(*!
<summary>Checks percentage dispersion for both signs and bound forwarding.</summary>
<description>
Owns a generator used by one PLC task. Each run checks the same bounds against fresh samples.
The runner binds assertions to the instance address. Keep the instance at that address for its run.
</description>
*)

{attribute 'no_assign'}
{attribute 'no_explicit_call' := 'do not call this function block directly'}
FUNCTION_BLOCK RandomPercentageDispersionTest EXTENDS TOF_Testing.SingleCycleTest
VAR_STAT
	{attribute 'hide'}
	_ClassName : STRING := __POUNAME();
END_VAR
VAR
	_Random : TOF_Core.Random;
END_VAR

(*!
<summary>Samples positive and negative bases and checks exact outcomes for zero and clamped dispersion.</summary>
<description>
The generated ranges have independently calculated endpoints. Enabled bounds cover deterministic cases
outside the generated interval. The test makes no assumptions about sample sequence or distribution.
</description>
*)
METHOD PROTECTED ExecuteTest
VAR
	value : LREAL;
	i : INT;
END_VAR
value := _Random.GetWithDispersionPercent(baseValue := LREAL#-40.0, dispersionPercent := LREAL#0.0);
Assert.ThatLongReal(
	actual := value,
	message := "Zero percent must return the negative base"
).ToBe(expected := LREAL#-40.0);

value := _Random.GetWithDispersionPercent(
	baseValue := LREAL#80.0,
	dispersionPercent := LREAL#25.0,
	minValue := LREAL#110.0
);
Assert.ThatLongReal(
	actual := value,
	message := "Percentage dispersion must forward the lower bound"
).ToBe(expected := LREAL#110.0);

value := _Random.GetWithDispersionPercent(
	baseValue := LREAL#-40.0,
	dispersionPercent := LREAL#25.0,
	maxValue := LREAL#-60.0
);
Assert.ThatLongReal(
	actual := value,
	message := "Percentage dispersion must forward the upper bound"
).ToBe(expected := LREAL#-60.0);

FOR i := 1 TO 21 DO
	value := _Random.GetWithDispersionPercent(baseValue := LREAL#80.0, dispersionPercent := LREAL#25.0);
	Assert.ThatLongReal(
		actual := value,
		message := "Positive base sample below 60"
	).IsGreaterThanOrEquals(expected := LREAL#60.0);
	Assert.ThatLongReal(
		actual := value,
		message := "Positive base sample above 100"
	).IsLessThanOrEquals(expected := LREAL#100.0);

	value := _Random.GetWithDispersionPercent(baseValue := LREAL#-40.0, dispersionPercent := LREAL#25.0);
	Assert.ThatLongReal(
		actual := value,
		message := "Negative base sample below -50"
	).IsGreaterThanOrEquals(expected := LREAL#-50.0);
	Assert.ThatLongReal(
		actual := value,
		message := "Negative base sample above -30"
	).IsLessThanOrEquals(expected := LREAL#-30.0);
END_FOR
END_METHOD

//! <summary>Borrows the concrete class name. Callers must not modify it.</summary>
{attribute 'monitoring' := 'call'}
PROPERTY ClassName : REFERENCE TO STRING
GET
ClassName REF= _ClassName;
END_GET
END_PROPERTY

//! <summary>Borrows the compiler-initialized namespace name. Callers must not modify it.</summary>
{attribute 'monitoring' := 'call'}
PROPERTY NamespaceName : REFERENCE TO STRING
GET
NamespaceName REF= CurrentNamespace.Name;
END_GET
END_PROPERTY

//! <summary>Reports the concrete instance size in bytes.</summary>
{attribute 'monitoring' := 'call'}
PROPERTY SelfSize : ULINT
GET
SelfSize := XSIZEOF(THIS^);
END_GET
END_PROPERTY

END_FUNCTION_BLOCK

// ---- Tests/Core/ExceptionTestGroup.TcPOU
(*
SPDX-FileCopyrightText: c 2026 Oleksandr Tiutyk <trofimich@gmail.com>
SPDX-License-Identifier: MIT
License: https://opensource.org/license/mit
*)

(*!
<summary>Groups exception transport, diagnostics, cloning and graph contract tests.</summary>
<description>
Owns the independent child instances and their fixed registration array. Use from one PLC task at a stable address.
</description>
*)

{attribute 'no_assign'}
{attribute 'no_explicit_call' := 'do not call this function block directly'}
FUNCTION_BLOCK ExceptionTestGroup EXTENDS TOF_Testing.TestGroup<12>
VAR_STAT
	{attribute 'hide'}
	_ClassName : STRING := __POUNAME();
END_VAR
VAR
	_NotImplemented : NotImplementedExceptionTest(name := "SimpleException", parent := THIS^);
	_StandardChain : StandardExceptionChainTest(name := "StandardExceptions", parent := THIS^);
	_Aggregate : AggregateExceptionPropagationTest(name := "AggregateException", parent := THIS^);
	_SavedFramework : SavedFrameworkExceptionRethrowTest(name := "RethrowSavedFrameworkException", parent := THIS^);
	_NativeRethrow : SystemExceptionRethrowTest(name := "RethrowSystemExceptionAfterFramework", parent := THIS^);
	_TimestampFormatting : ExceptionTimestampFormattingTest(name := "TimestampFormatting", parent := THIS^);
	_SystemTimestamp : SystemExceptionTimestampFormattingTest(
		name := "SystemExceptionTimestampFormatting",
		parent := THIS^
	);
	_SystemClone : SystemExceptionCloneTest(name := "SystemExceptionClone", parent := THIS^);
	_AggregateClone : AggregateExceptionCloneTest(name := "AggregateCloneLifetime", parent := THIS^);
	_ArgumentTypeClone : ArgumentTypeExceptionCloneTest(name := "ArgumentTypeCloneIdentity", parent := THIS^);
	_GraphRejection : ExceptionGraphRejectionTest(name := "GraphRejection", parent := THIS^);
	_BoundedMessage : AggregateExceptionBoundedMessageTest(name := "BoundedMessage", parent := THIS^);

	_Children : ARRAY [0.._ChildCount - 1] OF TOF_Testing.ITestElement :=
	[
		_NotImplemented,
		_StandardChain,
		_Aggregate,
		_SavedFramework,
		_NativeRethrow,
		_TimestampFormatting,
		_SystemTimestamp,
		_SystemClone,
		_AggregateClone,
		_ArgumentTypeClone,
		_GraphRejection,
		_BoundedMessage
	];
END_VAR

//! <summary>Borrows the fixed child array. Callers must not modify it.</summary>
{attribute 'monitoring' := 'call'}
PROPERTY Children : REFERENCE TO ARRAY [0.._ChildCount - 1] OF TOF_Testing.ITestElement
GET
Children REF= _Children;
END_GET
END_PROPERTY

//! <summary>Borrows the concrete class name. Callers must not modify it.</summary>
{attribute 'monitoring' := 'call'}
PROPERTY ClassName : REFERENCE TO STRING
GET
ClassName REF= _ClassName;
END_GET
END_PROPERTY

//! <summary>Borrows the compiler-initialized namespace name. Callers must not modify it.</summary>
{attribute 'monitoring' := 'call'}
PROPERTY NamespaceName : REFERENCE TO STRING
GET
NamespaceName REF= CurrentNamespace.Name;
END_GET
END_PROPERTY

//! <summary>Reports the concrete instance size in bytes.</summary>
{attribute 'monitoring' := 'call'}
PROPERTY SelfSize : ULINT
GET
SelfSize := XSIZEOF(THIS^);
END_GET
END_PROPERTY

END_FUNCTION_BLOCK

// ---- Tests/Core/NotImplementedExceptionTest.TcPOU
(*
SPDX-FileCopyrightText: c 2026 Oleksandr Tiutyk <trofimich@gmail.com>
SPDX-License-Identifier: MIT
License: https://opensource.org/license/mit
*)

(*!
<summary>Checks concrete exception transport and diagnostics for an unimplemented POU.</summary>
<description>
Uses one task and stays at a stable address while assertions are bound to this instance.
</description>
*)

{attribute 'no_assign'}
{attribute 'no_explicit_call' := 'do not call this function block directly'}
FUNCTION_BLOCK NotImplementedExceptionTest EXTENDS TOF_Testing.SingleCycleTest
VAR_STAT
	{attribute 'hide'}
	_ClassName : STRING := __POUNAME();
END_VAR

(*!
<summary>Checks concrete exception transport and diagnostics for an unimplemented POU.</summary>
<description>
Injects a fixed source location so the expected text and metadata are independent of this test's name.
</description>
*)
METHOD PROTECTED ExecuteTest
VAR
	exceptionCode : __SYSTEM.ExceptionCode;
	caught : TOF_Core.IException;
	typed : TOF_Core.INotImplementedException;
	message : TOF_Core.ERROR_MESSAGE;
END_VAR
// Raise one exception to exercise the transport from the facade to the catch.
__TRY
	TOF_Core.Exceptions.ThrowNotImplemented(
		sourceNamespaceName := 'Tests',
		sourceClassName := 'ExceptionFixture',
		sourcePOUName := 'UnimplementedOperation',
		sourcePosition := 'P1'
	);
__CATCH(exceptionCode)
	caught := TOF_Core.ExceptionManager.GetLastException(
		exceptionCode := exceptionCode,
		catchPointNamespaceName := NamespaceName,
		catchPointPOUName := __POUNAME(),
		catchPointPosition := __POSITION()
	);
__ENDTRY

IF NOT __QUERYINTERFACE(caught, typed) THEN
	RecordFailure(message := "ThrowNotImplemented must propagate NotImplementedException");
	RETURN;
END_IF

message := typed.GetMessage();
Assert.ThatBool(
	actual := message = "Program organization unit 'Tests.ExceptionFixture.UnimplementedOperation()' is not implemented",
	message := "NotImplementedException must name the supplied POU"
).IsTrue();
Assert.ThatBool(
	actual := typed.SourcePosition = 'P1',
	message := "NotImplementedException must preserve the throw position"
).IsTrue();
Assert.ThatBool(
	actual := typed.IsDynamicInstance,
	message := "Facade transport must yield a task-managed exception"
).IsTrue();
END_METHOD

//! <summary>Borrows the concrete class name. Callers must not modify it.</summary>
{attribute 'monitoring' := 'call'}
PROPERTY ClassName : REFERENCE TO STRING
GET
ClassName REF= _ClassName;
END_GET
END_PROPERTY

//! <summary>Borrows the compiler-initialized namespace name. Callers must not modify it.</summary>
{attribute 'monitoring' := 'call'}
PROPERTY NamespaceName : REFERENCE TO STRING
GET
NamespaceName REF= CurrentNamespace.Name;
END_GET
END_PROPERTY

//! <summary>Reports the concrete instance size in bytes.</summary>
{attribute 'monitoring' := 'call'}
PROPERTY SelfSize : ULINT
GET
SelfSize := XSIZEOF(THIS^);
END_GET
END_PROPERTY

END_FUNCTION_BLOCK

// ---- Tests/Core/StandardExceptionChainTest.TcPOU
(*
SPDX-FileCopyrightText: c 2026 Oleksandr Tiutyk <trofimich@gmail.com>
SPDX-License-Identifier: MIT
License: https://opensource.org/license/mit
*)

(*!
<summary>Checks the text, inner identity and root of a three-level standard exception chain.</summary>
<description>
Uses one task and stays at a stable address while assertions are bound to this instance.
</description>
*)

{attribute 'no_assign'}
{attribute 'no_explicit_call' := 'do not call this function block directly'}
FUNCTION_BLOCK StandardExceptionChainTest EXTENDS TOF_Testing.SingleCycleTest
VAR_STAT
	{attribute 'hide'}
	_ClassName : STRING := __POUNAME();
END_VAR

(*!
<summary>Checks the text, inner identity and root of a three-level standard exception chain.</summary>
<description>
Keeps only cycle-local references. Compares the root with the first caught cause through read-only views.
ToError copies the outer diagnostic and the deepest cause.
</description>
*)
METHOD PROTECTED ExecuteTest
VAR
	exceptionCode : __SYSTEM.ExceptionCode;
	caught : TOF_Core.IException;
	previous : TOF_Core.IException;
	previousView : TOF_Core.IReadOnlyException;
	first : TOF_Core.IReadOnlyException;
	root : TOF_Core.IReadOnlyException;
	typed : TOF_Core.IStandardException;

	inputs : ARRAY [0..2] OF WSTRING := ["First cause", "Second cause", "Outer failure"];
	expected : ARRAY [0..2] OF WSTRING := [
		"First cause",
		"Second cause -> First cause",
		"Outer failure -> Second cause -> First cause"
	];
	message : TOF_Core.ERROR_MESSAGE;
	actual : TOF_Core.ERROR_MESSAGE;
	snapshot : TOF_Core.ERROR;
	i : DINT;
END_VAR
FOR i := 0 TO UPPER_BOUND(inputs, 1) DO
	message := inputs[i];
	caught := 0;

	// Each deliberate throw adds one outer cause and is captured before asserting its payload.
	__TRY
		TOF_Core.Exceptions.ThrowStandard(
			sourceNamespaceName := NamespaceName,
			sourceClassName := ClassName,
			sourcePOUName := __POUNAME(),
			sourcePosition := __POSITION(),
			message := message,
			innerException := previous
		);
	__CATCH(exceptionCode)
		caught := TOF_Core.ExceptionManager.GetLastException(
			exceptionCode := exceptionCode,
			catchPointNamespaceName := NamespaceName,
			catchPointPOUName := __POUNAME(),
			catchPointPosition := __POSITION()
		);
	__ENDTRY

	IF NOT __QUERYINTERFACE(caught, typed) THEN
		Assert.ThatBool(
			actual := FALSE,
			message := Tc2_Utilities.WCONCAT(STR1 := "StandardException missing for ", STR2 := inputs[i])
		).IsTrue();
		RETURN;
	END_IF

	actual := typed.GetMessage();
	Assert.ThatBool(
		actual := actual = expected[i],
		message := Tc2_Utilities.WCONCAT(STR1 := "Incorrect chain text for ", STR2 := inputs[i])
	).IsTrue();
	Assert.ThatBool(
		actual := typed.InnerException = previousView,
		message := Tc2_Utilities.WCONCAT(STR1 := "Incorrect immediate cause for ", STR2 := inputs[i])
	).IsTrue();

	IF i = 0 THEN
		first := typed;
	END_IF

	previous := caught;
	previousView := typed;
END_FOR

root := typed.GetRootException();
Assert.ThatBool(
	actual := root = first,
	message := "The outer standard exception must reach the first cause"
).IsTrue();
typed.ToError(targetError := snapshot, severity := TOF_Core.ERROR_SEVERITY.CRITICAL);
Assert.ThatBool(
	actual := snapshot.TopMessage = expected[2] AND_THEN snapshot.RootMessage = "First cause",
	message := "The ERROR snapshot must keep the outer diagnostics and the deepest cause"
).IsTrue();
Assert.ThatBool(
	actual := snapshot.Severity = TOF_Core.ERROR_SEVERITY.CRITICAL,
	message := "ToError must copy the supplied severity"
).IsTrue();
END_METHOD

//! <summary>Borrows the concrete class name. Callers must not modify it.</summary>
{attribute 'monitoring' := 'call'}
PROPERTY ClassName : REFERENCE TO STRING
GET
ClassName REF= _ClassName;
END_GET
END_PROPERTY

//! <summary>Borrows the compiler-initialized namespace name. Callers must not modify it.</summary>
{attribute 'monitoring' := 'call'}
PROPERTY NamespaceName : REFERENCE TO STRING
GET
NamespaceName REF= CurrentNamespace.Name;
END_GET
END_PROPERTY

//! <summary>Reports the concrete instance size in bytes.</summary>
{attribute 'monitoring' := 'call'}
PROPERTY SelfSize : ULINT
GET
SelfSize := XSIZEOF(THIS^);
END_GET
END_PROPERTY

END_FUNCTION_BLOCK

// ---- Tests/Core/AggregateExceptionPropagationTest.TcPOU
(*
SPDX-FileCopyrightText: c 2026 Oleksandr Tiutyk <trofimich@gmail.com>
SPDX-License-Identifier: MIT
License: https://opensource.org/license/mit
*)

(*!
<summary>Checks aggregate flattening, transport, ordering and diagnostic snapshots.</summary>
<description>
Uses one task and stays at a stable address while assertions are bound to this instance.
</description>
*)

{attribute 'no_assign'}
{attribute 'no_explicit_call' := 'do not call this function block directly'}
FUNCTION_BLOCK AggregateExceptionPropagationTest EXTENDS TOF_Testing.SingleCycleTest
VAR_STAT
	{attribute 'hide'}
	_ClassName : STRING := __POUNAME();
END_VAR
VAR
	_Aggregate : TOF_Core.AggregateException;
	_AdditionalCauses : TOF_Core.AggregateException;
END_VAR

(*!
<summary>Checks aggregate flattening, transport, ordering and diagnostic snapshots.</summary>
<description>
The persistent arrays belong to this test. Within the current PLC cycle, compares borrowed causes by
read-only interface identity and checks null results on both sides of the valid index range.
Compares the full default message and reports the expected and actual text if they differ.
</description>
*)
METHOD PROTECTED ExecuteTest
VAR
	exceptionCode : __SYSTEM.ExceptionCode;
	caught : TOF_Core.IException;
	cause : TOF_Core.IStandardException;
	aggregate : TOF_Core.IAggregateException;
	causes : ARRAY [0..2] OF TOF_Core.IReadOnlyException;
	observedCause : TOF_Core.IReadOnlyException;

	causeMessages : ARRAY [0..2] OF WSTRING := ["First cause", "Second cause", "Third cause"];
	causeMessage : TOF_Core.ERROR_MESSAGE;
	message : TOF_Core.ERROR_MESSAGE;
	expectedMessage : TOF_Core.ERROR_MESSAGE;
	snapshot : TOF_Core.ERROR;
	i : DINT;
END_VAR
FOR i := 0 TO UPPER_BOUND(causes, 1) DO
	causeMessage := causeMessages[i];
	caught := 0;

	// Capture each deliberate throw before adding its task-owned payload to the fixture.
	__TRY
		TOF_Core.Exceptions.ThrowStandard(
			sourceNamespaceName := NamespaceName,
			sourceClassName := ClassName,
			sourcePOUName := 'RaiseCause',
			sourcePosition := __POSITION(),
			message := causeMessage
		);
	__CATCH(exceptionCode)
		caught := TOF_Core.ExceptionManager.GetLastException(
			exceptionCode := exceptionCode,
			catchPointNamespaceName := NamespaceName,
			catchPointPOUName := __POUNAME(),
			catchPointPosition := __POSITION()
		);
	__ENDTRY

	IF NOT __QUERYINTERFACE(caught, cause) THEN
		Assert.ThatBool(
			actual := FALSE,
			message := Tc2_Utilities.WCONCAT(STR1 := "Aggregate setup did not catch ", STR2 := causeMessages[i])
		).IsTrue();
		RETURN;
	END_IF

	causes[i] := cause;

	IF i = 0 THEN
		_Aggregate.AddInnerException(innerException := cause);
	ELSE
		_AdditionalCauses.AddInnerException(innerException := cause);
	END_IF
END_FOR

_Aggregate.AddInnerException(innerException := _AdditionalCauses);
_AdditionalCauses.Clear();

// Catch the aggregate snapshot before clearing its caller-owned source.
caught := 0;

__TRY
	_Aggregate.Throw(
		sourceNamespaceName := NamespaceName,
		sourceClassName := ClassName,
		sourcePOUName := __POUNAME(),
		sourcePosition := __POSITION()
	);
__CATCH(exceptionCode)
	caught := TOF_Core.ExceptionManager.GetLastException(
		exceptionCode := exceptionCode,
		catchPointNamespaceName := NamespaceName,
		catchPointPOUName := __POUNAME(),
		catchPointPosition := __POSITION()
	);
__ENDTRY

_Aggregate.Clear();

IF NOT __QUERYINTERFACE(caught, aggregate) THEN
	RecordFailure(message := "Aggregate Throw must propagate a concrete aggregate snapshot");
	RETURN;
END_IF

Assert.ThatUInt(
	actual := aggregate.InnerExceptionCount,
	message := "The propagated aggregate must contain all three flattened causes"
).ToBe(expected := UINT#3);

FOR i := 0 TO UPPER_BOUND(causes, 1) DO
	observedCause := aggregate.GetInnerException(index := i);
	Assert.ThatBool(
		actual := observedCause = causes[i],
		message := Tc2_Utilities.WCONCAT(STR1 := "Wrong aggregate position for ", STR2 := causeMessages[i])
	).IsTrue();
END_FOR

observedCause := aggregate.GetInnerException(index := -1);
Assert.ThatBool(
	actual := observedCause = 0,
	message := "Aggregate indexing before the first entry must return null"
).IsTrue();

observedCause := aggregate.GetInnerException(index := 3);
Assert.ThatBool(
	actual := observedCause = 0,
	message := "Aggregate indexing after the last entry must return null"
).IsTrue();

observedCause := aggregate.GetRootException();
Assert.ThatBool(
	actual := observedCause = causes[0],
	message := "Aggregate root must come from the first cause"
).IsTrue();

// The index suffix includes a space and the formatter appends one more before each cause.
expectedMessage := "3 aggregated exceptions$R0:  First cause$R1:  Second cause$R2:  Third cause";
message := aggregate.GetMessage();
Assert.That(
	actual := message,
	message := "The aggregate must describe all three causes in index order"
).ToBe(expected := expectedMessage);

aggregate.ToError(targetError := snapshot, severity := TOF_Core.ERROR_SEVERITY.CRITICAL);
Assert.ThatBool(
	actual := snapshot.TopMessage = message AND_THEN snapshot.RootMessage = "First cause",
	message := "The aggregate ERROR must copy the complete message and the first root diagnostic"
).IsTrue();
Assert.ThatBool(
	actual := snapshot.Severity = TOF_Core.ERROR_SEVERITY.CRITICAL,
	message := "Aggregate ToError must copy the supplied severity"
).IsTrue();
END_METHOD

(*!
<summary>Clears the caller-owned aggregate storage before the result is reported.</summary>
<description>
Safe after partial setup or repeated Clear. The task memory manager retains ownership of dynamic causes.
</description>
*)
METHOD PROTECTED AfterTest
_AdditionalCauses.Clear();
_Aggregate.Clear();
END_METHOD

//! <summary>Borrows the concrete class name. Callers must not modify it.</summary>
{attribute 'monitoring' := 'call'}
PROPERTY ClassName : REFERENCE TO STRING
GET
ClassName REF= _ClassName;
END_GET
END_PROPERTY

//! <summary>Borrows the compiler-initialized namespace name. Callers must not modify it.</summary>
{attribute 'monitoring' := 'call'}
PROPERTY NamespaceName : REFERENCE TO STRING
GET
NamespaceName REF= CurrentNamespace.Name;
END_GET
END_PROPERTY

//! <summary>Reports the concrete instance size in bytes.</summary>
{attribute 'monitoring' := 'call'}
PROPERTY SelfSize : ULINT
GET
SelfSize := XSIZEOF(THIS^);
END_GET
END_PROPERTY

END_FUNCTION_BLOCK

// ---- Tests/Core/SavedFrameworkExceptionRethrowTest.TcPOU
(*
SPDX-FileCopyrightText: c 2026 Oleksandr Tiutyk <trofimich@gmail.com>
SPDX-License-Identifier: MIT
License: https://opensource.org/license/mit
*)

(*!
<summary>Checks rethrow of a saved framework payload after a different nested exception.</summary>
<description>
Uses one task and stays at a stable address while assertions are bound to this instance.
</description>
*)

{attribute 'no_assign'}
{attribute 'no_explicit_call' := 'do not call this function block directly'}
FUNCTION_BLOCK SavedFrameworkExceptionRethrowTest EXTENDS TOF_Testing.SingleCycleTest
VAR_STAT
	{attribute 'hide'}
	_ClassName : STRING := __POUNAME();
END_VAR

(*!
<summary>Checks rethrow of a saved framework payload after a different nested exception.</summary>
<description>
The nested handler must capture its own payload. All caught references are used only in the current task cycle.
</description>
*)
METHOD PROTECTED ExecuteTest
VAR
	exceptionCode : __SYSTEM.ExceptionCode;
	saved : TOF_Core.IException;
	outerCode : __SYSTEM.ExceptionCode;
	nestedCode : __SYSTEM.ExceptionCode;
	nested : TOF_Core.IException;
	received : TOF_Core.IException;
	nestedMessage : TOF_Core.ERROR_MESSAGE;
	receivedMessage : TOF_Core.ERROR_MESSAGE;
END_VAR
// Catch the original, let a nested handler replace the active payload, then rethrow the saved object.
__TRY
	__TRY
		TOF_Core.Exceptions.ThrowStandard(
			sourceNamespaceName := NamespaceName,
			sourceClassName := ClassName,
			sourcePOUName := __POUNAME(),
			sourcePosition := __POSITION(),
			message := "Original"
		);
	__CATCH(exceptionCode)
		saved := TOF_Core.ExceptionManager.GetLastException(
			exceptionCode := exceptionCode,
			catchPointNamespaceName := NamespaceName,
			catchPointPOUName := __POUNAME(),
			catchPointPosition := __POSITION()
		);

		__TRY
			TOF_Core.Exceptions.ThrowStandard(
				sourceNamespaceName := NamespaceName,
				sourceClassName := ClassName,
				sourcePOUName := __POUNAME(),
				sourcePosition := __POSITION(),
				message := "Nested"
			);
		__CATCH(nestedCode)
			nested := TOF_Core.ExceptionManager.GetLastException(
				exceptionCode := nestedCode,
				catchPointNamespaceName := NamespaceName,
				catchPointPOUName := __POUNAME(),
				catchPointPosition := __POSITION()
			);
		__ENDTRY

		IF saved <> 0 THEN
			TOF_Core.ExceptionManager.Throw(exception := saved);
		END_IF
	__ENDTRY
__CATCH(outerCode)
	received := TOF_Core.ExceptionManager.GetLastException(
		exceptionCode := outerCode,
		catchPointNamespaceName := NamespaceName,
		catchPointPOUName := __POUNAME(),
		catchPointPosition := __POSITION()
	);
__ENDTRY

IF nested = 0 OR_ELSE received = 0 THEN
	RecordFailure(message := "The nested throw and the saved rethrow must both reach their handlers");
	RETURN;
END_IF

nestedMessage := nested.GetMessage();
receivedMessage := received.GetMessage();
Assert.ThatBool(
	actual := nested <> saved AND_THEN nestedMessage = "Nested",
	message := "The nested catch must observe a distinct payload"
).IsTrue();
Assert.ThatBool(
	actual := received = saved AND_THEN receivedMessage = "Original",
	message := "Rethrow must preserve the saved payload and text"
).IsTrue();
END_METHOD

//! <summary>Borrows the concrete class name. Callers must not modify it.</summary>
{attribute 'monitoring' := 'call'}
PROPERTY ClassName : REFERENCE TO STRING
GET
ClassName REF= _ClassName;
END_GET
END_PROPERTY

//! <summary>Borrows the compiler-initialized namespace name. Callers must not modify it.</summary>
{attribute 'monitoring' := 'call'}
PROPERTY NamespaceName : REFERENCE TO STRING
GET
NamespaceName REF= CurrentNamespace.Name;
END_GET
END_PROPERTY

//! <summary>Reports the concrete instance size in bytes.</summary>
{attribute 'monitoring' := 'call'}
PROPERTY SelfSize : ULINT
GET
SelfSize := XSIZEOF(THIS^);
END_GET
END_PROPERTY

END_FUNCTION_BLOCK

// ---- Tests/Core/SystemExceptionRethrowTest.TcPOU
(*
SPDX-FileCopyrightText: c 2026 Oleksandr Tiutyk <trofimich@gmail.com>
SPDX-License-Identifier: MIT
License: https://opensource.org/license/mit
*)

(*!
<summary>Checks native wrapper propagation through both framework rethrow APIs.</summary>
<description>
Uses one task and stays at a stable address while assertions are bound to this instance.
</description>
*)

{attribute 'no_assign'}
{attribute 'no_explicit_call' := 'do not call this function block directly'}
FUNCTION_BLOCK SystemExceptionRethrowTest EXTENDS TOF_Testing.SingleCycleTest
VAR_STAT
	{attribute 'hide'}
	_ClassName : STRING := __POUNAME();
END_VAR

(*!
<summary>Checks native wrapper propagation through both framework rethrow APIs.</summary>
<description>
Models captured native codes. A second native catch overwrites the shared wrapper while the propagated
snapshot retains its identity and payload until task cleanup.
</description>
*)
METHOD PROTECTED ExecuteTest
VAR
	exceptionCode : __SYSTEM.ExceptionCode;
	frameworkException : TOF_Core.IException;
	original : TOF_Core.IException;
	received : TOF_Core.IException;
	repeated : TOF_Core.IException;
	other : TOF_Core.IException;
	otherWrapper : TOF_Core.ISystemException;
	firstWrapper : TOF_Core.ISystemException;
	codeOnlyWrapper : TOF_Core.ISystemException;
	originalMessage : TOF_Core.ERROR_MESSAGE;
	message : TOF_Core.ERROR_MESSAGE;
	localTimestamp : LDATE_AND_TIME;
	utcTimestamp : LDATE_AND_TIME;
END_VAR
// Establish a framework payload before supplying an already received native code.
__TRY
	TOF_Core.Exceptions.ThrowStandard(
		sourceNamespaceName := NamespaceName,
		sourceClassName := ClassName,
		sourcePOUName := __POUNAME(),
		sourcePosition := __POSITION(),
		message := "Earlier framework payload"
	);
__CATCH(exceptionCode)
	frameworkException := TOF_Core.ExceptionManager.GetLastException(
		exceptionCode := exceptionCode,
		catchPointNamespaceName := NamespaceName,
		catchPointPOUName := __POUNAME(),
		catchPointPosition := __POSITION()
	);
__ENDTRY

IF frameworkException = 0 THEN
	RecordFailure(message := "The earlier framework throw must reach its handler");
	RETURN;
END_IF

original := TOF_Core.ExceptionManager.GetLastException(
	exceptionCode := __SYSTEM.ExceptionCode.RTSEXCPT_ARRAYBOUNDS,
	catchPointNamespaceName := 'Tests',
	catchPointPOUName := 'OriginalCatch',
	catchPointPosition := 'P1'
);

IF original = 0 THEN
	RecordFailure(message := "The captured native code must provide a wrapper");
	RETURN;
END_IF

originalMessage := original.GetMessage();
localTimestamp := original.LocalTimestamp;
utcTimestamp := original.UtcTimestamp;

// Transport the static native wrapper as a task-managed framework payload.
__TRY
	TOF_Core.ExceptionManager.Throw(exception := original);
__CATCH(exceptionCode)
	received := TOF_Core.ExceptionManager.GetLastException(
		exceptionCode := exceptionCode,
		catchPointNamespaceName := NamespaceName,
		catchPointPOUName := __POUNAME(),
		catchPointPosition := __POSITION()
	);
__ENDTRY

IF NOT __QUERYINTERFACE(received, firstWrapper) THEN
	RecordFailure(message := "Throw must preserve ISystemException after an earlier framework exception");
	RETURN;
END_IF

Assert.ThatBool(
	actual := firstWrapper.IsDynamicInstance AND_THEN received <> original,
	message := "Native propagation must clone the shared static wrapper"
).IsTrue();
Assert.ThatBool(
	actual := firstWrapper.ExceptionCode = __SYSTEM.ExceptionCode.RTSEXCPT_ARRAYBOUNDS,
	message := "The propagated wrapper must retain its captured native code"
).IsTrue();
Assert.ThatBool(
	actual := firstWrapper.LocalTimestamp = localTimestamp AND_THEN firstWrapper.UtcTimestamp = utcTimestamp,
	message := "Propagation must preserve both original timestamps"
).IsTrue();

other := TOF_Core.ExceptionManager.GetLastException(
	exceptionCode := __SYSTEM.ExceptionCode.RTSEXCPT_ACCESS_VIOLATION,
	catchPointNamespaceName := 'Tests',
	catchPointPOUName := 'OtherCatch',
	catchPointPosition := 'P2'
);
Assert.ThatBool(
	actual := other = original,
	message := "Another native catch must reuse the task wrapper"
).IsTrue();
Assert.ThatBool(
	actual := __QUERYINTERFACE(other, otherWrapper)
		AND_THEN otherWrapper.ExceptionCode = __SYSTEM.ExceptionCode.RTSEXCPT_ACCESS_VIOLATION,
	message := "The shared wrapper must actually observe the later native code"
).IsTrue();

message := firstWrapper.GetMessage();
Assert.ThatBool(
	actual := message = originalMessage
		AND_THEN Tc2_Standard.WFIND(STR1 := message, STR2 := "Tests.OriginalCatch at P1") > 0,
	message := "The propagated wrapper must keep its original diagnostic after the shared wrapper is overwritten"
).IsTrue();

// Replace the manager payload before rethrowing the saved dynamic wrapper.
frameworkException := 0;

__TRY
	TOF_Core.Exceptions.ThrowStandard(
		sourceNamespaceName := NamespaceName,
		sourceClassName := ClassName,
		sourcePOUName := __POUNAME(),
		sourcePosition := __POSITION(),
		message := "Intervening framework payload"
	);
__CATCH(exceptionCode)
	frameworkException := TOF_Core.ExceptionManager.GetLastException(
		exceptionCode := exceptionCode,
		catchPointNamespaceName := NamespaceName,
		catchPointPOUName := __POUNAME(),
		catchPointPosition := __POSITION()
	);
__ENDTRY

Assert.ThatBool(
	actual := frameworkException <> 0 AND_THEN frameworkException <> received,
	message := "An intervening framework throw must install a different payload"
).IsTrue();

__TRY
	TOF_Core.ExceptionManager.Throw(exception := received);
__CATCH(exceptionCode)
	repeated := TOF_Core.ExceptionManager.GetLastException(
		exceptionCode := exceptionCode,
		catchPointNamespaceName := NamespaceName,
		catchPointPOUName := __POUNAME(),
		catchPointPosition := __POSITION()
	);
__ENDTRY

Assert.ThatBool(
	actual := repeated = received,
	message := "Rethrowing the dynamic wrapper must preserve its identity"
).IsTrue();

// Exercise callers that pass a native code and catch point instead of keeping a payload.
repeated := 0;

__TRY
	TOF_Core.ExceptionManager.ReThrowLastException(
		exceptionCode := __SYSTEM.ExceptionCode.RTSEXCPT_ARRAYBOUNDS,
		catchPointNamespaceName := 'Tests',
		catchPointPOUName := 'OriginalCatch',
		catchPointPosition := 'P1'
	);
__CATCH(exceptionCode)
	repeated := TOF_Core.ExceptionManager.GetLastException(
		exceptionCode := exceptionCode,
		catchPointNamespaceName := NamespaceName,
		catchPointPOUName := __POUNAME(),
		catchPointPosition := __POSITION()
	);
__ENDTRY

IF NOT __QUERYINTERFACE(repeated, codeOnlyWrapper) THEN
	RecordFailure(message := "Code-only rethrow must provide an ISystemException payload");
	RETURN;
END_IF

message := codeOnlyWrapper.GetMessage();
Assert.ThatBool(
	actual := message = originalMessage,
	message := "Code-only rethrow must retain the supplied native diagnostic and location"
).IsTrue();
Assert.ThatBool(
	actual := codeOnlyWrapper.ExceptionCode = __SYSTEM.ExceptionCode.RTSEXCPT_ARRAYBOUNDS,
	message := "Code-only rethrow must preserve the native code"
).IsTrue();
END_METHOD

//! <summary>Borrows the concrete class name. Callers must not modify it.</summary>
{attribute 'monitoring' := 'call'}
PROPERTY ClassName : REFERENCE TO STRING
GET
ClassName REF= _ClassName;
END_GET
END_PROPERTY

//! <summary>Borrows the compiler-initialized namespace name. Callers must not modify it.</summary>
{attribute 'monitoring' := 'call'}
PROPERTY NamespaceName : REFERENCE TO STRING
GET
NamespaceName REF= CurrentNamespace.Name;
END_GET
END_PROPERTY

//! <summary>Reports the concrete instance size in bytes.</summary>
{attribute 'monitoring' := 'call'}
PROPERTY SelfSize : ULINT
GET
SelfSize := XSIZEOF(THIS^);
END_GET
END_PROPERTY

END_FUNCTION_BLOCK

// ---- Tests/Core/ExceptionTimestampFormattingTest.TcPOU
(*
SPDX-FileCopyrightText: c 2026 Oleksandr Tiutyk <trofimich@gmail.com>
SPDX-License-Identifier: MIT
License: https://opensource.org/license/mit
*)

(*!
<summary>Checks the shared exception timestamp formatter with fixed local and UTC inputs.</summary>
<description>
Uses one task and stays at a stable address while assertions are bound to this instance.
</description>
*)

{attribute 'no_assign'}
{attribute 'no_explicit_call' := 'do not call this function block directly'}
FUNCTION_BLOCK ExceptionTimestampFormattingTest EXTENDS TOF_Testing.SingleCycleTest
VAR_STAT
	{attribute 'hide'}
	_ClassName : STRING := __POUNAME();
END_VAR
VAR
	_Probe : ExceptionTimestampProbe;
END_VAR

(*!
<summary>Checks the shared exception timestamp formatter with fixed local and UTC inputs.</summary>
<description>
Calls the existing adapter with deterministic timestamps. The result uses the exception diagnostic capacity.
</description>
*)
METHOD PROTECTED ExecuteTest
VAR
	message : TOF_Core.ERROR_MESSAGE;
END_VAR
VAR CONSTANT
	LOCAL_TIMESTAMP : LDATE_AND_TIME := LDT#2026-10-06-15:04:05;
	UTC_TIMESTAMP : LDATE_AND_TIME := LDT#2026-10-06-12:04:05;
END_VAR
message := _Probe.FormatTimestamp(
	mode := TOF_Core.TIMESTAMP_DISPLAY_MODE.HIDDEN,
	localTime := LOCAL_TIMESTAMP,
	utcTime := UTC_TIMESTAMP
);
Assert.ThatBool(
	actual := message = "",
	message := "Hidden timestamp must leave an empty target unchanged"
).IsTrue();

message := _Probe.FormatTimestamp(
	mode := TOF_Core.TIMESTAMP_DISPLAY_MODE.LOCAL,
	localTime := LOCAL_TIMESTAMP,
	utcTime := UTC_TIMESTAMP
);
Assert.ThatBool(
	actual := Tc2_Standard.WFIND(STR1 := message, STR2 := "15:04:05") > 0,
	message := "LOCAL formatting must use local time"
).IsTrue();
Assert.ThatBool(
	actual := Tc2_Standard.WFIND(STR1 := message, STR2 := "UTC") = 0,
	message := "LOCAL formatting must omit the UTC suffix"
).IsTrue();

message := _Probe.FormatTimestamp(
	mode := TOF_Core.TIMESTAMP_DISPLAY_MODE.UTC,
	localTime := LOCAL_TIMESTAMP,
	utcTime := UTC_TIMESTAMP
);
Assert.ThatBool(
	actual := Tc2_Standard.WFIND(STR1 := message, STR2 := "12:04:05") > 0,
	message := "UTC formatting must use UTC time"
).IsTrue();
Assert.ThatBool(
	actual := Tc2_Standard.WRIGHT(STR := message, SIZE := 3) = "UTC",
	message := "UTC formatting must retain the UTC suffix"
).IsTrue();
END_METHOD

//! <summary>Borrows the concrete class name. Callers must not modify it.</summary>
{attribute 'monitoring' := 'call'}
PROPERTY ClassName : REFERENCE TO STRING
GET
ClassName REF= _ClassName;
END_GET
END_PROPERTY

//! <summary>Borrows the compiler-initialized namespace name. Callers must not modify it.</summary>
{attribute 'monitoring' := 'call'}
PROPERTY NamespaceName : REFERENCE TO STRING
GET
NamespaceName REF= CurrentNamespace.Name;
END_GET
END_PROPERTY

//! <summary>Reports the concrete instance size in bytes.</summary>
{attribute 'monitoring' := 'call'}
PROPERTY SelfSize : ULINT
GET
SelfSize := XSIZEOF(THIS^);
END_GET
END_PROPERTY

END_FUNCTION_BLOCK

// ---- Tests/Core/ExceptionTimestampProbe.TcPOU
(*
SPDX-FileCopyrightText: © 2026 Oleksandr Tiutyk <trofimich@gmail.com>
SPDX-License-Identifier: MIT
License: https://opensource.org/license/mit
*)

(*!
<summary>Static test adapter exposing the inherited formatter with deterministic inputs.</summary>
*)

FUNCTION_BLOCK ExceptionTimestampProbe EXTENDS TOF_Core.StandardException

METHOD FormatTimestamp : TOF_Core.ERROR_MESSAGE
VAR_INPUT
	mode : TOF_Core.TIMESTAMP_DISPLAY_MODE;
	localTime : LDATE_AND_TIME;
	utcTime : LDATE_AND_TIME;
END_VAR
AppendTimestampDescription(
	targetMessage := FormatTimestamp,
	timestampDisplayMode := mode,
	localTimestamp := localTime,
	utcTimestamp := utcTime
);
END_METHOD

END_FUNCTION_BLOCK

// ---- Tests/Core/SystemExceptionTimestampFormattingTest.TcPOU
(*
SPDX-FileCopyrightText: c 2026 Oleksandr Tiutyk <trofimich@gmail.com>
SPDX-License-Identifier: MIT
License: https://opensource.org/license/mit
*)

(*!
<summary>Checks the native wrapper message in HIDDEN, LOCAL and UTC modes.</summary>
<description>
Uses one task and stays at a stable address while assertions are bound to this instance.
</description>
*)

{attribute 'no_assign'}
{attribute 'no_explicit_call' := 'do not call this function block directly'}
FUNCTION_BLOCK SystemExceptionTimestampFormattingTest EXTENDS TOF_Testing.SingleCycleTest
VAR_STAT
	{attribute 'hide'}
	_ClassName : STRING := __POUNAME();
END_VAR

(*!
<summary>Checks the native wrapper message in HIDDEN, LOCAL and UTC modes.</summary>
<description>
Uses the borrowed wrapper during one callback. The timestamp expectations use the IEC conversion of
captured values and a separately assembled expected message.
</description>
*)
METHOD PROTECTED ExecuteTest
VAR
	exception : TOF_Core.IException;
	hidden : TOF_Core.ERROR_MESSAGE;
	message : TOF_Core.ERROR_MESSAGE;
	expected : WSTRING(255);
	formattingFailed : BOOL;
END_VAR
exception := TOF_Core.ExceptionManager.GetLastException(
	exceptionCode := __SYSTEM.ExceptionCode.RTSEXCPT_ACCESS_VIOLATION,
	catchPointNamespaceName := 'TimestampTest',
	catchPointPOUName := 'NativeCatch',
	catchPointPosition := 'P1'
);

IF exception = 0 THEN
	RecordFailure(message := "The captured native code must provide a wrapper");
	RETURN;
END_IF

hidden := exception.GetMessage(timestampDisplayMode := TOF_Core.TIMESTAMP_DISPLAY_MODE.HIDDEN);
Assert.ThatBool(
	actual := Tc2_Standard.WRIGHT(STR := hidden, SIZE := 31) = "TimestampTest.NativeCatch at P1",
	message := "The hidden timestamp mode must end with the supplied catch location"
).IsTrue();

expected := Tc2_Utilities.WCONCAT(STR1 := hidden, STR2 := " at ");
expected := Tc2_Utilities.WCONCAT(STR1 := expected, STR2 := TO_WSTRING(exception.LocalTimestamp));
formattingFailed := FALSE;

// A formatter exception is recorded for this mode before proceeding to the next check.
__TRY
	message := exception.GetMessage(timestampDisplayMode := TOF_Core.TIMESTAMP_DISPLAY_MODE.LOCAL);
__CATCH
	formattingFailed := TRUE;
__ENDTRY

Assert.ThatBool(
	actual := NOT formattingFailed AND_THEN message = expected,
	message := "LOCAL must append its captured timestamp"
).IsTrue();

expected := Tc2_Utilities.WCONCAT(STR1 := hidden, STR2 := " at ");
expected := Tc2_Utilities.WCONCAT(STR1 := expected, STR2 := TO_WSTRING(exception.UtcTimestamp));
expected := Tc2_Utilities.WCONCAT(STR1 := expected, STR2 := "UTC");
formattingFailed := FALSE;

// A formatter exception is recorded for this mode before proceeding to the next check.
__TRY
	message := exception.GetMessage(timestampDisplayMode := TOF_Core.TIMESTAMP_DISPLAY_MODE.UTC);
__CATCH
	formattingFailed := TRUE;
__ENDTRY

Assert.ThatBool(
	actual := NOT formattingFailed AND_THEN message = expected,
	message := "UTC must append its captured timestamp and UTC suffix"
).IsTrue();

message := exception.GetMessage(timestampDisplayMode := TOF_Core.TIMESTAMP_DISPLAY_MODE.HIDDEN);
Assert.ThatBool(
	actual := message = hidden,
	message := "Timestamp formatting must preserve the underlying diagnostic"
).IsTrue();
END_METHOD

//! <summary>Borrows the concrete class name. Callers must not modify it.</summary>
{attribute 'monitoring' := 'call'}
PROPERTY ClassName : REFERENCE TO STRING
GET
ClassName REF= _ClassName;
END_GET
END_PROPERTY

//! <summary>Borrows the compiler-initialized namespace name. Callers must not modify it.</summary>
{attribute 'monitoring' := 'call'}
PROPERTY NamespaceName : REFERENCE TO STRING
GET
NamespaceName REF= CurrentNamespace.Name;
END_GET
END_PROPERTY

//! <summary>Reports the concrete instance size in bytes.</summary>
{attribute 'monitoring' := 'call'}
PROPERTY SelfSize : ULINT
GET
SelfSize := XSIZEOF(THIS^);
END_GET
END_PROPERTY

END_FUNCTION_BLOCK

// ---- Tests/Core/SystemExceptionCloneTest.TcPOU
(*
SPDX-FileCopyrightText: c 2026 Oleksandr Tiutyk <trofimich@gmail.com>
SPDX-License-Identifier: MIT
License: https://opensource.org/license/mit
*)

(*!
<summary>Checks a direct clone before and after the task-local system wrapper is reconfigured.</summary>
<description>
Uses one task and stays at a stable address while assertions are bound to this instance.
</description>
*)

{attribute 'no_assign'}
{attribute 'no_explicit_call' := 'do not call this function block directly'}
FUNCTION_BLOCK SystemExceptionCloneTest EXTENDS TOF_Testing.SingleCycleTest
VAR_STAT
	{attribute 'hide'}
	_ClassName : STRING := __POUNAME();
END_VAR

(*!
<summary>Checks a direct clone before and after the task-local system wrapper is reconfigured.</summary>
<description>
Supplies native codes to the adapter without raising a native exception. The clone is valid until task cleanup.
</description>
*)
METHOD PROTECTED ExecuteTest
VAR
	original : TOF_Core.IException;
	reconfigured : TOF_Core.IException;
	clonedObject : TOF_Core.IObject;
	cloned : TOF_Core.ISystemException;
	expected : TOF_Core.ERROR_MESSAGE;
	actual : TOF_Core.ERROR_MESSAGE;
	localTimestamp : LDATE_AND_TIME;
	utcTimestamp : LDATE_AND_TIME;
END_VAR
original := TOF_Core.ExceptionManager.GetLastException(
	exceptionCode := __SYSTEM.ExceptionCode.RTSEXCPT_OUT_OF_MEMORY,
	catchPointNamespaceName := 'CloneTest',
	catchPointPOUName := 'OriginalCatch',
	catchPointPosition := 'P1'
);

IF original = 0 THEN
	RecordFailure(message := "The native code must produce a shared wrapper");
	RETURN;
END_IF

expected := original.GetMessage();
localTimestamp := original.LocalTimestamp;
utcTimestamp := original.UtcTimestamp;
clonedObject := original.Clone();

IF NOT __QUERYINTERFACE(clonedObject, cloned) THEN
	RecordFailure(message := "A SystemException clone must implement ISystemException");
	RETURN;
END_IF

Assert.ThatBool(
	actual := cloned.IsDynamicInstance AND_THEN cloned.SelfAddress <> original.SelfAddress,
	message := "The clone must be a distinct task-managed instance"
).IsTrue();

reconfigured := TOF_Core.ExceptionManager.GetLastException(
	exceptionCode := __SYSTEM.ExceptionCode.RTSEXCPT_NOEXCEPTION,
	catchPointNamespaceName := 'Changed',
	catchPointPOUName := 'Changed',
	catchPointPosition := 'P2'
);
Assert.ThatBool(
	actual := reconfigured = original AND_THEN original.Empty,
	message := "The same shared wrapper must be empty after reconfiguration"
).IsTrue();
Assert.ThatBool(
	actual := cloned.ExceptionCode = __SYSTEM.ExceptionCode.RTSEXCPT_OUT_OF_MEMORY,
	message := "The clone must retain the captured native code"
).IsTrue();

actual := cloned.GetMessage();
Assert.ThatBool(
	actual := actual = expected AND_THEN Tc2_Standard.WFIND(STR1 := actual, STR2 := "CloneTest.OriginalCatch at P1") > 0,
	message := "The clone must retain the original diagnostic and catch location"
).IsTrue();
Assert.ThatBool(
	actual := cloned.LocalTimestamp = localTimestamp AND_THEN cloned.UtcTimestamp = utcTimestamp,
	message := "The clone must retain both captured timestamps"
).IsTrue();
END_METHOD

//! <summary>Borrows the concrete class name. Callers must not modify it.</summary>
{attribute 'monitoring' := 'call'}
PROPERTY ClassName : REFERENCE TO STRING
GET
ClassName REF= _ClassName;
END_GET
END_PROPERTY

//! <summary>Borrows the compiler-initialized namespace name. Callers must not modify it.</summary>
{attribute 'monitoring' := 'call'}
PROPERTY NamespaceName : REFERENCE TO STRING
GET
NamespaceName REF= CurrentNamespace.Name;
END_GET
END_PROPERTY

//! <summary>Reports the concrete instance size in bytes.</summary>
{attribute 'monitoring' := 'call'}
PROPERTY SelfSize : ULINT
GET
SelfSize := XSIZEOF(THIS^);
END_GET
END_PROPERTY

END_FUNCTION_BLOCK

// ---- Tests/Core/AggregateExceptionCloneTest.TcPOU
(*
SPDX-FileCopyrightText: c 2026 Oleksandr Tiutyk <trofimich@gmail.com>
SPDX-License-Identifier: MIT
License: https://opensource.org/license/mit
*)

(*!
<summary>Checks that an aggregate clone owns its array and shares its prepared dynamic causes.</summary>
<description>
Uses one task and stays at a stable address while assertions are bound to this instance.
</description>
*)

{attribute 'no_assign'}
{attribute 'no_explicit_call' := 'do not call this function block directly'}
FUNCTION_BLOCK AggregateExceptionCloneTest EXTENDS TOF_Testing.SingleCycleTest
VAR_STAT
	{attribute 'hide'}
	_ClassName : STRING := __POUNAME();
END_VAR
VAR
	_Aggregate : TOF_Core.AggregateException;
END_VAR

(*!
<summary>Checks that an aggregate clone owns its array and shares its prepared dynamic causes.</summary>
<description>
The source is persistent so AfterTest can release its array after an unexpected hook exception.
Checks identity through borrowed read-only interfaces during the current task cycle.
</description>
*)
METHOD PROTECTED ExecuteTest
VAR
	exceptionCode : __SYSTEM.ExceptionCode;
	caught : TOF_Core.IException;
	source : TOF_Core.StandardException;
	dynamicInner : TOF_Core.IReadOnlyException;
	staticSource : TOF_Core.IReadOnlyException;
	firstInner : TOF_Core.IReadOnlyException;
	observedInner : TOF_Core.IReadOnlyException;
	clonedObject : TOF_Core.IObject;
	clonedAggregate : TOF_Core.IAggregateException;
	message : TOF_Core.ERROR_MESSAGE;
END_VAR
// Throwing the static template provides a dynamic cause with the same initial message.
__TRY
	source.Throw(
		sourceNamespaceName := NamespaceName,
		sourceClassName := ClassName,
		sourcePOUName := __POUNAME(),
		sourcePosition := __POSITION(),
		message := "Original inner"
	);
__CATCH(exceptionCode)
	caught := TOF_Core.ExceptionManager.GetLastException(
		exceptionCode := exceptionCode,
		catchPointNamespaceName := NamespaceName,
		catchPointPOUName := __POUNAME(),
		catchPointPosition := __POSITION()
	);
__ENDTRY

IF caught = 0 THEN
	RecordFailure(message := "Throw must provide a dynamic cause for the clone test");
	RETURN;
END_IF

Assert.ThatBool(
	actual := caught.IsDynamicInstance,
	message := "The thrown cause must belong to task cleanup"
).IsTrue();

staticSource := source;
dynamicInner := caught;
_Aggregate.AddInnerException(innerException := staticSource);
_Aggregate.AddInnerException(innerException := dynamicInner);
source.Clear();

firstInner := _Aggregate.GetInnerException(index := 0);

IF firstInner = 0 THEN
	RecordFailure(message := "The aggregate must store the prepared clone of the static cause");
	RETURN;
END_IF

message := firstInner.GetMessage();
Assert.ThatBool(
	actual := firstInner <> staticSource AND_THEN message = "Original inner",
	message := "The static cause must be cloned before its template is cleared"
).IsTrue();
observedInner := _Aggregate.GetInnerException(index := 1);
Assert.ThatBool(
	actual := observedInner = dynamicInner,
	message := "The dynamic cause must retain its identity"
).IsTrue();

clonedObject := _Aggregate.Clone();
_Aggregate.Clear();
_Aggregate.Clear();
Assert.ThatBool(
	actual := _Aggregate.Empty AND_THEN _Aggregate.InnerExceptionCount = 0,
	message := "Repeated Clear must leave the original aggregate empty"
).IsTrue();

IF NOT __QUERYINTERFACE(clonedObject, clonedAggregate) THEN
	RecordFailure(message := "Aggregate clone must preserve its concrete interface");
	RETURN;
END_IF

Assert.ThatBool(
	actual := clonedAggregate.IsDynamicInstance AND_THEN clonedAggregate.SelfAddress <> _Aggregate.SelfAddress,
	message := "The aggregate clone must be a distinct task-managed instance"
).IsTrue();
Assert.ThatUInt(
	actual := clonedAggregate.InnerExceptionCount,
	message := "Clearing the original must preserve the clone's array"
).ToBe(expected := UINT#2);

observedInner := clonedAggregate.GetInnerException(index := 0);
Assert.ThatBool(
	actual := observedInner = firstInner,
	message := "The clone must share the prepared first cause"
).IsTrue();

observedInner := clonedAggregate.GetInnerException(index := 1);
Assert.ThatBool(
	actual := observedInner = dynamicInner,
	message := "The clone must share the second dynamic cause"
).IsTrue();
END_METHOD

(*!
<summary>Clears the caller-owned aggregate storage before the result is reported.</summary>
<description>
Safe after partial setup or repeated Clear. The task memory manager retains ownership of dynamic causes.
</description>
*)
METHOD PROTECTED AfterTest
_Aggregate.Clear();
END_METHOD

//! <summary>Borrows the concrete class name. Callers must not modify it.</summary>
{attribute 'monitoring' := 'call'}
PROPERTY ClassName : REFERENCE TO STRING
GET
ClassName REF= _ClassName;
END_GET
END_PROPERTY

//! <summary>Borrows the compiler-initialized namespace name. Callers must not modify it.</summary>
{attribute 'monitoring' := 'call'}
PROPERTY NamespaceName : REFERENCE TO STRING
GET
NamespaceName REF= CurrentNamespace.Name;
END_GET
END_PROPERTY

//! <summary>Reports the concrete instance size in bytes.</summary>
{attribute 'monitoring' := 'call'}
PROPERTY SelfSize : ULINT
GET
SelfSize := XSIZEOF(THIS^);
END_GET
END_PROPERTY

END_FUNCTION_BLOCK

// ---- Tests/Core/ArgumentTypeExceptionCloneTest.TcPOU
(*
SPDX-FileCopyrightText: c 2026 Oleksandr Tiutyk <trofimich@gmail.com>
SPDX-License-Identifier: MIT
License: https://opensource.org/license/mit
*)

(*!
<summary>Checks concrete identity and copied fields of a populated argument-type exception clone.</summary>
<description>
Uses one task and stays at a stable address while assertions are bound to this instance.
</description>
*)

{attribute 'no_assign'}
{attribute 'no_explicit_call' := 'do not call this function block directly'}
FUNCTION_BLOCK ArgumentTypeExceptionCloneTest EXTENDS TOF_Testing.SingleCycleTest
VAR_STAT
	{attribute 'hide'}
	_ClassName : STRING := __POUNAME();
END_VAR

(*!
<summary>Checks concrete identity and copied fields of a populated argument-type exception clone.</summary>
<description>
Copies the configured source within the current task cycle. Clears the source before reading the registered clone.
</description>
*)
METHOD PROTECTED ExecuteTest
VAR
	exceptionCode : __SYSTEM.ExceptionCode;
	caught : TOF_Core.IException;
	source : TOF_Core.ArgumentTypeNotSupportedException;
	thrown : TOF_Core.IArgumentTypeNotSupportedException;
	clonedObject : TOF_Core.IObject;
	cloned : TOF_Core.IArgumentTypeNotSupportedException;
	localTimestamp : LDATE_AND_TIME;
	utcTimestamp : LDATE_AND_TIME;
END_VAR
// Configure the source through its normal Throw API and catch the resulting framework payload.
__TRY
	source.Throw(
		sourceNamespaceName := 'Tests',
		sourceClassName := 'ArgumentFixture',
		sourcePOUName := 'Reject',
		sourcePosition := 'P1',
		argumentName := 'value',
		argumentTypeName := 'UNSUPPORTED_TYPE'
	);
__CATCH(exceptionCode)
	caught := TOF_Core.ExceptionManager.GetLastException(
		exceptionCode := exceptionCode,
		catchPointNamespaceName := NamespaceName,
		catchPointPOUName := __POUNAME(),
		catchPointPosition := __POSITION()
	);
__ENDTRY

IF NOT __QUERYINTERFACE(caught, thrown) THEN
	RecordFailure(message := "ArgumentTypeNotSupportedException must preserve its type on Throw");
	RETURN;
END_IF

localTimestamp := source.LocalTimestamp;
utcTimestamp := source.UtcTimestamp;
clonedObject := source.Clone();
source.Clear();

IF NOT __QUERYINTERFACE(clonedObject, cloned) THEN
	RecordFailure(message := "Clone must implement IArgumentTypeNotSupportedException");
	RETURN;
END_IF

Assert.ThatBool(
	actual := cloned.IsDynamicInstance AND_THEN cloned.SelfAddress <> source.SelfAddress,
	message := "The clone must be distinct from the caller-owned template"
).IsTrue();
Assert.ThatBool(
	actual := cloned.SourceMessage
		= "Argument 'value' has not supported type 'UNSUPPORTED_TYPE' in 'Tests.ArgumentFixture.Reject()'",
	message := "The clone must preserve the argument name, unsupported type and POU"
).IsTrue();
Assert.ThatBool(
	actual := cloned.SourceFullPOUName = 'Tests.ArgumentFixture.Reject()' AND_THEN cloned.SourcePosition = 'P1',
	message := "The clone must preserve its original source metadata"
).IsTrue();
Assert.ThatBool(
	actual := cloned.LocalTimestamp = localTimestamp AND_THEN cloned.UtcTimestamp = utcTimestamp,
	message := "The clone must preserve both occurrence timestamps"
).IsTrue();
END_METHOD

//! <summary>Borrows the concrete class name. Callers must not modify it.</summary>
{attribute 'monitoring' := 'call'}
PROPERTY ClassName : REFERENCE TO STRING
GET
ClassName REF= _ClassName;
END_GET
END_PROPERTY

//! <summary>Borrows the compiler-initialized namespace name. Callers must not modify it.</summary>
{attribute 'monitoring' := 'call'}
PROPERTY NamespaceName : REFERENCE TO STRING
GET
NamespaceName REF= CurrentNamespace.Name;
END_GET
END_PROPERTY

//! <summary>Reports the concrete instance size in bytes.</summary>
{attribute 'monitoring' := 'call'}
PROPERTY SelfSize : ULINT
GET
SelfSize := XSIZEOF(THIS^);
END_GET
END_PROPERTY

END_FUNCTION_BLOCK

// ---- Tests/Core/ExceptionGraphRejectionTest.TcPOU
(*
SPDX-FileCopyrightText: c 2026 Oleksandr Tiutyk <trofimich@gmail.com>
SPDX-License-Identifier: MIT
License: https://opensource.org/license/mit
*)

(*!
<summary>Checks that aggregate and standard exceptions reject a direct self-reference before mutation.</summary>
<description>
Uses one task and stays at a stable address while assertions are bound to this instance.
</description>
*)

{attribute 'no_assign'}
{attribute 'no_explicit_call' := 'do not call this function block directly'}
FUNCTION_BLOCK ExceptionGraphRejectionTest EXTENDS TOF_Testing.SingleCycleTest
VAR_STAT
	{attribute 'hide'}
	_ClassName : STRING := __POUNAME();
END_VAR
VAR
	_Aggregate : TOF_Core.AggregateException;
END_VAR

(*!
<summary>Checks that aggregate and standard exceptions reject a direct self-reference before mutation.</summary>
<description>
Uses caller-owned objects and captures each expected rejection in the same PLC cycle.
</description>
*)
METHOD PROTECTED ExecuteTest
VAR
	exceptionCode : __SYSTEM.ExceptionCode;
	caught : TOF_Core.IException;
	typed : TOF_Core.IStandardException;
	source : TOF_Core.StandardException;
END_VAR
// This insertion would introduce a cycle. The test only reads the count after the attempted insertion.
__TRY
	_Aggregate.AddInnerException(innerException := _Aggregate);
__CATCH(exceptionCode)
	caught := TOF_Core.ExceptionManager.GetLastException(
		exceptionCode := exceptionCode,
		catchPointNamespaceName := NamespaceName,
		catchPointPOUName := __POUNAME(),
		catchPointPosition := __POSITION()
	);
__ENDTRY

IF NOT __QUERYINTERFACE(caught, typed) THEN
	RecordFailure(message := "Attaching an aggregate to itself must raise StandardException");
	RETURN;
END_IF

Assert.ThatBool(
	actual := typed.SourceMessage = "Cannot attach an exception graph containing its prospective owner."
	AND_THEN typed.InnerException = 0,
	message := "Aggregate cycle rejection must report the graph error without an inner cause"
).IsTrue();
Assert.ThatBool(
	actual := _Aggregate.InnerExceptionCount = 0,
	message := "Rejected attachment must preserve the empty aggregate"
).IsTrue();

caught := 0;

// Populate a standard template so a failed self-attachment can be checked for partial mutation.
__TRY
	source.Throw(
		sourceNamespaceName := NamespaceName,
		sourceClassName := ClassName,
		sourcePOUName := __POUNAME(),
		sourcePosition := 'ExistingPosition',
		message := "Existing message"
	);
__CATCH(exceptionCode)
	caught := TOF_Core.ExceptionManager.GetLastException(
		exceptionCode := exceptionCode,
		catchPointNamespaceName := NamespaceName,
		catchPointPOUName := __POUNAME(),
		catchPointPosition := __POSITION()
	);
__ENDTRY

IF NOT __QUERYINTERFACE(caught, typed) THEN
	RecordFailure(message := "The standard template must be initialized by the deliberate throw");
	RETURN;
END_IF
Assert.ThatBool(
	actual := source.SourceMessage = "Existing message",
	message := "The standard template must start with the expected message"
).IsTrue();

caught := 0;

// Attempt to attach the caller-owned template to itself.
__TRY
	source.Throw(
		sourceNamespaceName := NamespaceName,
		sourceClassName := ClassName,
		sourcePOUName := __POUNAME(),
		sourcePosition := 'ReplacementPosition',
		message := "Replacement message",
		innerException := source
	);
__CATCH(exceptionCode)
	caught := TOF_Core.ExceptionManager.GetLastException(
		exceptionCode := exceptionCode,
		catchPointNamespaceName := NamespaceName,
		catchPointPOUName := __POUNAME(),
		catchPointPosition := __POSITION()
	);
__ENDTRY

IF NOT __QUERYINTERFACE(caught, typed) THEN
	RecordFailure(message := "Attaching a standard exception to itself must raise StandardException");
	RETURN;
END_IF

Assert.ThatBool(
	actual := typed.SourceMessage = "Cannot attach an exception graph containing its prospective owner."
	AND_THEN typed.InnerException = 0,
	message := "Standard cycle rejection must report the graph error without an inner cause"
).IsTrue();
Assert.ThatBool(
	actual := source.SourceMessage = "Existing message"
	AND_THEN source.SourcePosition = 'ExistingPosition'
	AND_THEN source.InnerException = 0,
	message := "Rejected attachment must preserve the original standard exception fields"
).IsTrue();
END_METHOD

(*!
<summary>Clears the caller-owned aggregate storage before the result is reported.</summary>
<description>
Safe after partial setup or repeated Clear. The task memory manager retains ownership of dynamic causes.
</description>
*)
METHOD PROTECTED AfterTest
_Aggregate.Clear();
END_METHOD

//! <summary>Borrows the concrete class name. Callers must not modify it.</summary>
{attribute 'monitoring' := 'call'}
PROPERTY ClassName : REFERENCE TO STRING
GET
ClassName REF= _ClassName;
END_GET
END_PROPERTY

//! <summary>Borrows the compiler-initialized namespace name. Callers must not modify it.</summary>
{attribute 'monitoring' := 'call'}
PROPERTY NamespaceName : REFERENCE TO STRING
GET
NamespaceName REF= CurrentNamespace.Name;
END_GET
END_PROPERTY

//! <summary>Reports the concrete instance size in bytes.</summary>
{attribute 'monitoring' := 'call'}
PROPERTY SelfSize : ULINT
GET
SelfSize := XSIZEOF(THIS^);
END_GET
END_PROPERTY

END_FUNCTION_BLOCK

// ---- Tests/Core/AggregateExceptionBoundedMessageTest.TcPOU
(*
SPDX-FileCopyrightText: c 2026 Oleksandr Tiutyk <trofimich@gmail.com>
SPDX-License-Identifier: MIT
License: https://opensource.org/license/mit
*)

(*!
<summary>Checks that a long aggregate diagnostic is terminated and ends in an ellipsis.</summary>
<description>
Uses one task and stays at a stable address while assertions are bound to this instance.
</description>
*)

{attribute 'no_assign'}
{attribute 'no_explicit_call' := 'do not call this function block directly'}
FUNCTION_BLOCK AggregateExceptionBoundedMessageTest EXTENDS TOF_Testing.SingleCycleTest
VAR_STAT
	{attribute 'hide'}
	_ClassName : STRING := __POUNAME();
END_VAR
VAR
	_Aggregate : TOF_Core.AggregateException;
END_VAR

(*!
<summary>Checks that a long aggregate diagnostic is terminated and ends in an ellipsis.</summary>
<description>
Three entries share one task-managed cause. Each payload fills half the diagnostic buffer so the
combined message exceeds its capacity. The persistent reference array is released in AfterTest.
</description>
*)
METHOD PROTECTED ExecuteTest
VAR
	exceptionCode : __SYSTEM.ExceptionCode;
	caught : TOF_Core.IException;
	cause : TOF_Core.IStandardException;
	payload : TOF_Core.ERROR_MESSAGE;
	message : TOF_Core.ERROR_MESSAGE;
	payloadUnits : POINTER TO WORD;
	messageUnits : POINTER TO WORD;
	i : UDINT;
END_VAR
VAR CONSTANT
	MESSAGE_CAPACITY : UDINT := TOF_Core.Parameters.ERROR_MESSAGE_WIDE_CHAR_SIZE;
END_VAR
// Make an ASCII payload whose length scales with the documented diagnostic capacity.
payloadUnits := ADR(payload);

FOR i := 0 TO MESSAGE_CAPACITY / 2 - 1 DO
	payloadUnits[i] := WORD#16#0058; // Uppercase X makes the retained prefix distinguishable from the ellipsis.
END_FOR

payloadUnits[MESSAGE_CAPACITY / 2] := TO_WORD(TOF_Core.UnsignedInt16.MIN_VALUE);

// Obtain one dynamic cause so repeated entries exercise permitted sharing.
__TRY
	TOF_Core.Exceptions.ThrowStandard(
		sourceNamespaceName := NamespaceName,
		sourceClassName := ClassName,
		sourcePOUName := __POUNAME(),
		sourcePosition := __POSITION(),
		message := payload
	);
__CATCH(exceptionCode)
	caught := TOF_Core.ExceptionManager.GetLastException(
		exceptionCode := exceptionCode,
		catchPointNamespaceName := NamespaceName,
		catchPointPOUName := __POUNAME(),
		catchPointPosition := __POSITION()
	);
__ENDTRY

IF NOT __QUERYINTERFACE(caught, cause) THEN
	RecordFailure(message := "A task-owned payload is required for the aggregate length check");
	RETURN;
END_IF

_Aggregate.AddInnerException(innerException := cause);
_Aggregate.AddInnerException(innerException := cause);
_Aggregate.AddInnerException(innerException := cause);
message := _Aggregate.GetMessage();

messageUnits := ADR(message);

IF messageUnits[MESSAGE_CAPACITY] <> TO_WORD(TOF_Core.UnsignedInt16.MIN_VALUE) THEN
	RecordFailure(message := "The last storage unit must terminate the aggregate diagnostic");
	RETURN;
END_IF

Assert.ThatUDInt(
	actual := TOF_Core.WideStrings.GetLength(value := message),
	message := "The bounded aggregate message must fill the available character capacity"
).ToBe(expected := MESSAGE_CAPACITY);
Assert.ThatBool(
	actual := Tc2_Standard.WFIND(STR1 := message, STR2 := "3 aggregated exceptions$R0:") = 1,
	message := "The bounded message must retain the aggregate header and the first entry marker"
).IsTrue();
Assert.ThatBool(
	actual := messageUnits[MESSAGE_CAPACITY - 2] = WORD#16#0058,
	message := "The bounded message must retain cause text immediately before the ellipsis"
).IsTrue();
Assert.ThatBool(
	actual := messageUnits[MESSAGE_CAPACITY - 1] = TOF_Core.WideStrings.ELLIPSIS,
	message := "The final character must be an ellipsis"
).IsTrue();
END_METHOD

(*!
<summary>Clears the caller-owned aggregate storage before the result is reported.</summary>
<description>
Safe after partial setup or repeated Clear. The task memory manager retains ownership of dynamic causes.
</description>
*)
METHOD PROTECTED AfterTest
_Aggregate.Clear();
END_METHOD

//! <summary>Borrows the concrete class name. Callers must not modify it.</summary>
{attribute 'monitoring' := 'call'}
PROPERTY ClassName : REFERENCE TO STRING
GET
ClassName REF= _ClassName;
END_GET
END_PROPERTY

//! <summary>Borrows the compiler-initialized namespace name. Callers must not modify it.</summary>
{attribute 'monitoring' := 'call'}
PROPERTY NamespaceName : REFERENCE TO STRING
GET
NamespaceName REF= CurrentNamespace.Name;
END_GET
END_PROPERTY

//! <summary>Reports the concrete instance size in bytes.</summary>
{attribute 'monitoring' := 'call'}
PROPERTY SelfSize : ULINT
GET
SelfSize := XSIZEOF(THIS^);
END_GET
END_PROPERTY

END_FUNCTION_BLOCK

// ---- Tests/Strings/String/StringsTestGroup.TcPOU
(*
SPDX-FileCopyrightText: c 2026 Oleksandr Tiutyk <trofimich@gmail.com>
SPDX-License-Identifier: MIT
License: https://opensource.org/license/mit
*)

(*!
<summary>Groups byte-string formatting, editing, search and splitter contracts.</summary>
<description>
Owns the independent child instances and their fixed registration array. Use from one PLC task at a stable address.
</description>
*)

{attribute 'no_assign'}
{attribute 'no_explicit_call' := 'do not call this function block directly'}
FUNCTION_BLOCK StringsTestGroup EXTENDS TOF_Testing.TestGroup<10>
VAR_STAT
	{attribute 'hide'}
	_ClassName : STRING := __POUNAME();
END_VAR
VAR
	_AnyToStringFit255 : StringFitFormattingTest(name := "AnyToStringFit255", parent := THIS^);
	_Append : StringAppendTest(name := "Append", parent := THIS^);
	_AppendFit : StringAppendFitTest(name := "AppendFit", parent := THIS^);
	_ConcatFit255 : StringConcatFitTest(name := "ConcatFit255", parent := THIS^);
	_Contains : StringContainsTest(name := "Contains", parent := THIS^);
	_Join : StringJoinTest(name := "Join", parent := THIS^);
	_ReplaceInSource : StringReplacementTest(name := "ReplaceInSource", parent := THIS^);
	_Split : StringSplitTest(name := "Split", parent := THIS^);
	_Trim : StringTrimTest(name := "Trim", parent := THIS^);
	_SplitterSeparatorBounds : StringSeparatorBoundsTest(name := "SplitterSeparatorBounds", parent := THIS^);

	_Children : ARRAY [0.._ChildCount - 1] OF TOF_Testing.ITestElement :=
	[
		_AnyToStringFit255,
		_Append,
		_AppendFit,
		_ConcatFit255,
		_Contains,
		_Join,
		_ReplaceInSource,
		_Split,
		_Trim,
		_SplitterSeparatorBounds
	];
END_VAR

//! <summary>Borrows the fixed child array. Callers must not modify it.</summary>
{attribute 'monitoring' := 'call'}
PROPERTY Children : REFERENCE TO ARRAY [0.._ChildCount - 1] OF TOF_Testing.ITestElement
GET
Children REF= _Children;
END_GET
END_PROPERTY

//! <summary>Borrows the concrete class name. Callers must not modify it.</summary>
{attribute 'monitoring' := 'call'}
PROPERTY ClassName : REFERENCE TO STRING
GET
ClassName REF= _ClassName;
END_GET
END_PROPERTY

//! <summary>Borrows the compiler-initialized namespace name. Callers must not modify it.</summary>
{attribute 'monitoring' := 'call'}
PROPERTY NamespaceName : REFERENCE TO STRING
GET
NamespaceName REF= CurrentNamespace.Name;
END_GET
END_PROPERTY

//! <summary>Reports the concrete instance size in bytes.</summary>
{attribute 'monitoring' := 'call'}
PROPERTY SelfSize : ULINT
GET
SelfSize := XSIZEOF(THIS^);
END_GET
END_PROPERTY

END_FUNCTION_BLOCK

// ---- Tests/Strings/String/StringFitFormattingTest.TcPOU
(*
SPDX-FileCopyrightText: c 2026 Oleksandr Tiutyk <trofimich@gmail.com>
SPDX-License-Identifier: MIT
License: https://opensource.org/license/mit
*)

(*!
<summary>Checks scalar and short text formatting through the fitted ANY API.</summary>
<description>
Uses one task and stays at a stable address while assertions are bound to this instance.
</description>
*)

{attribute 'no_assign'}
{attribute 'no_explicit_call' := 'do not call this function block directly'}
FUNCTION_BLOCK StringFitFormattingTest EXTENDS TOF_Testing.SingleCycleTest
VAR_STAT
	{attribute 'hide'}
	_ClassName : STRING := __POUNAME();
END_VAR

(*!
<summary>Checks scalar and short text formatting through the fitted ANY API.</summary>
<description>
Compares the complete results for a 255-byte ASCII input and a 256-byte ASCII input requiring truncation.
</description>
*)
METHOD PROTECTED ExecuteTest
VAR
	formatted : STRING(255);
	enabled : BOOL := TRUE;
	number : DINT := 12345;
	narrowText : STRING(50) := 'Sample string';
	wideText : WSTRING(50) := "Sample wide string";
	longText : STRING(256);
	textBytes : POINTER TO BYTE;
END_VAR
formatted := TOF_Core.Strings.AnyToStringFit255(value := enabled);
Assert.ThatBool(
	actual := formatted = 'TRUE',
	message := "AnyToStringFit255 must format BOOL"
).IsTrue();

formatted := TOF_Core.Strings.AnyToStringFit255(value := number);
Assert.ThatBool(
	actual := formatted = '12345',
	message := "AnyToStringFit255 must format DINT"
).IsTrue();

formatted := TOF_Core.Strings.AnyToStringFit255(value := narrowText);
Assert.ThatBool(
	actual := formatted = 'Sample string',
	message := "AnyToStringFit255 must pass short STRING as-is"
).IsTrue();

formatted := TOF_Core.Strings.AnyToStringFit255(value := wideText);
Assert.ThatBool(
	actual := formatted = 'Sample wide string',
	message := "AnyToStringFit255 must convert short WSTRING to STRING"
).IsTrue();

// SA0175: Use byte offsets for a bounded ASCII fixture of known size.
{analysis -175}
textBytes := ADR(longText);
{analysis +175}
Tc2_System.MEMSET(destAddr := textBytes, fillByte := BYTE#16#61, n := 255);
textBytes[255] := TO_BYTE(TOF_Core.UnsignedInt8.MIN_VALUE);
textBytes[256] := TO_BYTE(TOF_Core.UnsignedInt8.MIN_VALUE);

formatted := TOF_Core.Strings.AnyToStringFit255(value := longText);
Assert.ThatBool(
	actual := Tc2_Standard.LEN(STR := formatted) = 255 AND_THEN formatted = longText,
	message := "An exact-fit STRING must preserve all 255 bytes"
).IsTrue();

textBytes[255] := BYTE#16#61;
formatted := TOF_Core.Strings.AnyToStringFit255(value := longText);

// Form the expected output independently with 252 ASCII letters followed by three periods.
Tc2_System.MEMSET(destAddr := textBytes + 252, fillByte := BYTE#16#2E, n := 3);
textBytes[255] := TO_BYTE(TOF_Core.UnsignedInt8.MIN_VALUE);
Assert.ThatBool(
	actual := Tc2_Standard.LEN(STR := formatted) = 255 AND_THEN formatted = longText,
	message := "A 256-byte STRING must retain 252 bytes and append three dots"
).IsTrue();
END_METHOD

//! <summary>Borrows the concrete class name. Callers must not modify it.</summary>
{attribute 'monitoring' := 'call'}
PROPERTY ClassName : REFERENCE TO STRING
GET
ClassName REF= _ClassName;
END_GET
END_PROPERTY

//! <summary>Borrows the compiler-initialized namespace name. Callers must not modify it.</summary>
{attribute 'monitoring' := 'call'}
PROPERTY NamespaceName : REFERENCE TO STRING
GET
NamespaceName REF= CurrentNamespace.Name;
END_GET
END_PROPERTY

//! <summary>Reports the concrete instance size in bytes.</summary>
{attribute 'monitoring' := 'call'}
PROPERTY SelfSize : ULINT
GET
SelfSize := XSIZEOF(THIS^);
END_GET
END_PROPERTY

END_FUNCTION_BLOCK

// ---- Tests/Strings/String/StringAppendTest.TcPOU
(*
SPDX-FileCopyrightText: c 2026 Oleksandr Tiutyk <trofimich@gmail.com>
SPDX-License-Identifier: MIT
License: https://opensource.org/license/mit
*)

(*!
<summary>Checks strict and Try appends, including empty fragments and capacity failure.</summary>
<description>
Uses one task and stays at a stable address while assertions are bound to this instance.
</description>
*)

{attribute 'no_assign'}
{attribute 'no_explicit_call' := 'do not call this function block directly'}
FUNCTION_BLOCK StringAppendTest EXTENDS TOF_Testing.SingleCycleTest
VAR_STAT
	{attribute 'hide'}
	_ClassName : STRING := __POUNAME();
END_VAR

(*!
<summary>Checks strict and Try appends, including empty fragments and capacity failure.</summary>
<description>
Uses an eight-byte ASCII target. After a later fragment fails to fit, checks that the original text and the
first appended fragment remain at the start of the target.
</description>
*)
METHOD PROTECTED ExecuteTest
VAR
	target : STRING(8);
	accepted : BOOL;
	prefixFound : BOOL;
	prefixPosition : UDINT;
END_VAR
target := 'ab';
TOF_Core.Strings.Append255(target, 'cd', '', 'efgh');
Assert.ThatBool(
	actual := target = 'abcdefgh',
	message := "Append255 must skip an empty fragment and fill the target exactly"
).IsTrue();

target := 'ab';
accepted := TOF_Core.Strings.TryAppend255(
	targetString := target,
	sourceString1 := 'cd',
	sourceString2 := '',
	sourceString3 := 'efgh'
);
Assert.ThatBool(
	actual := accepted AND_THEN target = 'abcdefgh',
	message := "TryAppend255 must accept an exact fit"
).IsTrue();

target := 'ab';
accepted := TOF_Core.Strings.TryAppend255(
	targetString := target,
	sourceString1 := 'cd',
	sourceString2 := 'ABCDE',
	sourceString3 := '!'
);
Assert.ThatBool(
	actual := accepted,
	message := "TryAppend255 must report capacity failure"
).IsFalse();

prefixFound := TOF_Core.Strings.Find(
	stringToSearchIn := target,
	stringToFind := 'abcd',
	position => prefixPosition
);
Assert.ThatBool(
	actual := prefixFound AND_THEN prefixPosition = 1,
	message := "TryAppend255 must preserve the successfully appended prefix"
).IsTrue();

target := 'ab';
TOF_Core.Strings.Append(targetString := target, sourceString := 'cd');
TOF_Core.Strings.Append(targetString := target, sourceString := '');
TOF_Core.Strings.Append(targetString := target, sourceString := 'efgh');
Assert.ThatBool(
	actual := target = 'abcdefgh',
	message := "Append must preserve the target on empty input and accept the exact fit"
).IsTrue();

target := 'abcdef';
accepted := TOF_Core.Strings.TryAppend(targetString := target, sourceString := 'gh');
Assert.ThatBool(
	actual := accepted AND_THEN target = 'abcdefgh',
	message := "TryAppend must accept an exact fit"
).IsTrue();

accepted := TOF_Core.Strings.TryAppend(targetString := target, sourceString := 'i');
Assert.ThatBool(
	actual := accepted,
	message := "TryAppend must reject another character in a full target"
).IsFalse();
Assert.ThatBool(
	actual := target = 'abcdefgh',
	message := "TryAppend must preserve the full target when one more character does not fit"
).IsTrue();
END_METHOD

//! <summary>Borrows the concrete class name. Callers must not modify it.</summary>
{attribute 'monitoring' := 'call'}
PROPERTY ClassName : REFERENCE TO STRING
GET
ClassName REF= _ClassName;
END_GET
END_PROPERTY

//! <summary>Borrows the compiler-initialized namespace name. Callers must not modify it.</summary>
{attribute 'monitoring' := 'call'}
PROPERTY NamespaceName : REFERENCE TO STRING
GET
NamespaceName REF= CurrentNamespace.Name;
END_GET
END_PROPERTY

//! <summary>Reports the concrete instance size in bytes.</summary>
{attribute 'monitoring' := 'call'}
PROPERTY SelfSize : ULINT
GET
SelfSize := XSIZEOF(THIS^);
END_GET
END_PROPERTY

END_FUNCTION_BLOCK

// ---- Tests/Strings/String/StringAppendFitTest.TcPOU
(*
SPDX-FileCopyrightText: c 2026 Oleksandr Tiutyk <trofimich@gmail.com>
SPDX-License-Identifier: MIT
License: https://opensource.org/license/mit
*)

(*!
<summary>Checks fitted appends at exact capacity and on truncation.</summary>
<description>
Uses one task and stays at a stable address while assertions are bound to this instance.
</description>
*)

{attribute 'no_assign'}
{attribute 'no_explicit_call' := 'do not call this function block directly'}
FUNCTION_BLOCK StringAppendFitTest EXTENDS TOF_Testing.SingleCycleTest
VAR_STAT
	{attribute 'hide'}
	_ClassName : STRING := __POUNAME();
END_VAR

(*!
<summary>Checks fitted appends at exact capacity and on truncation.</summary>
*)
METHOD PROTECTED ExecuteTest
VAR
	oneCharacter : STRING(1);
	twoCharacters : STRING(2);
	target : STRING(10);
	longFragment : STRING(30) := '01234567890123456789';
	accepted : BOOL;
END_VAR
// Fits within capacity
target := '12345';
TOF_Core.Strings.AppendFit(targetString := target, sourceString := '67');
Assert.ThatBool(
	actual := target = '1234567',
	message := "AppendFit must append normally when it fits"
).IsTrue();

// Exact fit: fills capacity without ellipsis
target := '12345';
TOF_Core.Strings.AppendFit(targetString := target, sourceString := '67890');
Assert.ThatBool(
	actual := target = '1234567890',
	message := "AppendFit must fit exactly without ellipsis"
).IsTrue();

// Overflow by 1 char: truncates and appends '...'
target := '12345';
TOF_Core.Strings.AppendFit(targetString := target, sourceString := '678901');
Assert.ThatBool(
	actual := target = '1234567...',
	message := "AppendFit must truncate and append ... on 1 char overflow"
).IsTrue();

// Overflow by many chars: truncates and appends '...'
target := '12345';
TOF_Core.Strings.AppendFit(targetString := target, sourceString := longFragment);
Assert.ThatBool(
	actual := target = '1234501...',
	message := "AppendFit must truncate and append ... on large overflow"
).IsTrue();

// Empty source: target remains unchanged
target := '12345';
TOF_Core.Strings.AppendFit(targetString := target, sourceString := '');
Assert.ThatBool(
	actual := target = '12345',
	message := "AppendFit must leave target unchanged for empty source"
).IsTrue();

// Appending to empty target
target := '';
TOF_Core.Strings.AppendFit(targetString := target, sourceString := longFragment);
Assert.ThatBool(
	actual := target = '0123456...',
	message := "AppendFit to empty target must truncate and append ..."
).IsTrue();

// TryAppendFit normal fit
target := '123';
accepted := TOF_Core.Strings.TryAppendFit(targetString := target, sourceString := '45');
Assert.ThatBool(
	actual := accepted,
	message := "TryAppendFit must return TRUE on normal fit"
).IsTrue();
Assert.ThatBool(
	actual := target = '12345',
	message := "TryAppendFit must append text"
).IsTrue();

// TryAppendFit overflow
target := '12345';
accepted := TOF_Core.Strings.TryAppendFit(targetString := target, sourceString := longFragment);
Assert.ThatBool(
	actual := accepted,
	message := "TryAppendFit must return TRUE on overflow"
).IsTrue();
Assert.ThatBool(
	actual := target = '1234501...',
	message := "TryAppendFit must truncate and append ..."
).IsTrue();

// AppendFit255 multiple arguments and literals
target := '12';
TOF_Core.Strings.AppendFit255(target, '3', '4', '5');
Assert.ThatBool(
	actual := target = '12345',
	message := "AppendFit255 must append multiple fragments"
).IsTrue();

// AppendFit255 overflow truncation
target := '12';
TOF_Core.Strings.AppendFit255(target, '345', '678', '9012');
Assert.ThatBool(
	actual := target = '1234567...',
	message := "AppendFit255 must truncate and append ... on overflow"
).IsTrue();

// TryAppendFit255 normal fit
target := '12';
accepted := TOF_Core.Strings.TryAppendFit255(
	targetString := target,
	sourceString1 := '3',
	sourceString2 := '4',
	sourceString3 := '5'
);
Assert.ThatBool(
	actual := accepted,
	message := "TryAppendFit255 must return TRUE on normal fit"
).IsTrue();
Assert.ThatBool(
	actual := target = '12345',
	message := "TryAppendFit255 must append multiple fragments"
).IsTrue();

// TryAppendFit255 overflow
target := '12';
accepted := TOF_Core.Strings.TryAppendFit255(
	targetString := target,
	sourceString1 := '345',
	sourceString2 := '678',
	sourceString3 := '9012'
);
Assert.ThatBool(
	actual := accepted,
	message := "TryAppendFit255 must return TRUE on overflow"
).IsTrue();
Assert.ThatBool(
	actual := target = '1234567...',
	message := "TryAppendFit255 must truncate and append ... on overflow"
).IsTrue();

accepted := TOF_Core.Strings.TryAppendFit(targetString := oneCharacter, sourceString := longFragment);
Assert.ThatBool(
	actual := accepted,
	message := "Truncation must succeed in a one-character buffer"
).IsTrue();
Assert.ThatBool(
	actual := oneCharacter = '.',
	message := "One-character truncation marker"
).IsTrue();

accepted := TOF_Core.Strings.TryAppendFit255(targetString := twoCharacters, sourceString1 := longFragment);
Assert.ThatBool(
	actual := accepted,
	message := "Truncation must succeed in a two-character buffer"
).IsTrue();
Assert.ThatBool(
	actual := twoCharacters = '.',
	message := "Two-character truncation marker"
).IsTrue();
END_METHOD

//! <summary>Borrows the concrete class name. Callers must not modify it.</summary>
{attribute 'monitoring' := 'call'}
PROPERTY ClassName : REFERENCE TO STRING
GET
ClassName REF= _ClassName;
END_GET
END_PROPERTY

//! <summary>Borrows the compiler-initialized namespace name. Callers must not modify it.</summary>
{attribute 'monitoring' := 'call'}
PROPERTY NamespaceName : REFERENCE TO STRING
GET
NamespaceName REF= CurrentNamespace.Name;
END_GET
END_PROPERTY

//! <summary>Reports the concrete instance size in bytes.</summary>
{attribute 'monitoring' := 'call'}
PROPERTY SelfSize : ULINT
GET
SelfSize := XSIZEOF(THIS^);
END_GET
END_PROPERTY

END_FUNCTION_BLOCK

// ---- Tests/Strings/String/StringConcatFitTest.TcPOU
(*
SPDX-FileCopyrightText: c 2026 Oleksandr Tiutyk <trofimich@gmail.com>
SPDX-License-Identifier: MIT
License: https://opensource.org/license/mit
*)

(*!
<summary>Checks fitted concatenation, including the 255-character boundary.</summary>
<description>
Uses one task and stays at a stable address while assertions are bound to this instance.
</description>
*)

{attribute 'no_assign'}
{attribute 'no_explicit_call' := 'do not call this function block directly'}
FUNCTION_BLOCK StringConcatFitTest EXTENDS TOF_Testing.SingleCycleTest
VAR_STAT
	{attribute 'hide'}
	_ClassName : STRING := __POUNAME();
END_VAR

(*!
<summary>Checks fitted concatenation, including the 255-character boundary.</summary>
<description>
Distinct ASCII fragments reveal the first discarded byte and any changes in fragment order. Compares all
255 bytes against a separately assembled expected result.
</description>
*)
METHOD PROTECTED ExecuteTest
VAR
	text : STRING(255);
	first : STRING(100) := 'aaaaaaaaaaaaaaaaaaaaaaaaaaaaaaaaaaaaaaaaaaaaaaaaaaaaaaaaaaaaaaaaaaaaaaaaaaaaaaaaaaaaaaaaaaaaaaaaaaaa';
	second : STRING(100) := 'bbbbbbbbbbbbbbbbbbbbbbbbbbbbbbbbbbbbbbbbbbbbbbbbbbbbbbbbbbbbbbbbbbbbbbbbbbbbbbbbbbbbbbbbbbbbbbbbbbbb';
	third : STRING(100) := 'cccccccccccccccccccccccccccccccccccccccccccccccccccccccccccccccccccccccccccccccccccccccccccccccccccc';
	expectedText : STRING(255);
END_VAR
text := TOF_Core.Strings.ConcatFit255('Hello, ', 'World!');
Assert.ThatBool(
	actual := text = 'Hello, World!',
	message := "ConcatFit255 must preserve an ordinary fit"
).IsTrue();

text := TOF_Core.Strings.ConcatFit255('Part1', '', 'Part2', '', 'Part3');
Assert.ThatBool(
	actual := text = 'Part1Part2Part3',
	message := "ConcatFit255 must skip empty fragments without stopping"
).IsTrue();

text := TOF_Core.Strings.ConcatFit255(first, second, third);
Assert.ThatInt(
	actual := Tc2_Standard.LEN(STR := text),
	message := "ConcatFit255 must fill the 255-character result"
).ToBe(expected := 255);

// The first two 100-byte fragments leave room for 52 bytes from the third and the three-dot suffix.
expectedText := Tc2_Standard.CONCAT(STR1 := first, STR2 := second);
expectedText := Tc2_Standard.CONCAT(
	STR1 := expectedText,
	STR2 := 'cccccccccccccccccccccccccccccccccccccccccccccccccccc...'
);
Assert.ThatBool(
	actual := text = expectedText,
	message := "Truncation must preserve the 252-byte prefix and end in three dots"
).IsTrue();
END_METHOD

//! <summary>Borrows the concrete class name. Callers must not modify it.</summary>
{attribute 'monitoring' := 'call'}
PROPERTY ClassName : REFERENCE TO STRING
GET
ClassName REF= _ClassName;
END_GET
END_PROPERTY

//! <summary>Borrows the compiler-initialized namespace name. Callers must not modify it.</summary>
{attribute 'monitoring' := 'call'}
PROPERTY NamespaceName : REFERENCE TO STRING
GET
NamespaceName REF= CurrentNamespace.Name;
END_GET
END_PROPERTY

//! <summary>Reports the concrete instance size in bytes.</summary>
{attribute 'monitoring' := 'call'}
PROPERTY SelfSize : ULINT
GET
SelfSize := XSIZEOF(THIS^);
END_GET
END_PROPERTY

END_FUNCTION_BLOCK

// ---- Tests/Strings/String/StringContainsTest.TcPOU
(*
SPDX-FileCopyrightText: c 2026 Oleksandr Tiutyk <trofimich@gmail.com>
SPDX-License-Identifier: MIT
License: https://opensource.org/license/mit
*)

(*!
<summary>Checks exact, case-sensitive substring matching and empty inputs.</summary>
<description>
Uses one task and stays at a stable address while assertions are bound to this instance.
</description>
*)

{attribute 'no_assign'}
{attribute 'no_explicit_call' := 'do not call this function block directly'}
FUNCTION_BLOCK StringContainsTest EXTENDS TOF_Testing.SingleCycleTest
VAR_STAT
	{attribute 'hide'}
	_ClassName : STRING := __POUNAME();
END_VAR

(*!
<summary>Checks exact, case-sensitive substring matching and empty inputs.</summary>
*)
METHOD PROTECTED ExecuteTest
VAR
	containsResult : BOOL;
END_VAR
containsResult := TOF_Core.Strings.Contains(stringToSearchIn := 'Hello, world!', stringToFind := 'Hello');
Assert.ThatBool(
	actual := containsResult,
	message := "Contains must return TRUE for prefix substring"
).IsTrue();

containsResult := TOF_Core.Strings.Contains(stringToSearchIn := 'Hello, world!', stringToFind := 'world');
Assert.ThatBool(
	actual := containsResult,
	message := "Contains must return TRUE for middle substring"
).IsTrue();

containsResult := TOF_Core.Strings.Contains(stringToSearchIn := 'Hello, world!', stringToFind := '!');
Assert.ThatBool(
	actual := containsResult,
	message := "Contains must return TRUE for suffix substring"
).IsTrue();

containsResult := TOF_Core.Strings.Contains(stringToSearchIn := 'Hello, world!', stringToFind := 'Hello, world!');
Assert.ThatBool(
	actual := containsResult,
	message := "Contains must return TRUE for identical string"
).IsTrue();

containsResult := TOF_Core.Strings.Contains(stringToSearchIn := 'Hello, world!', stringToFind := '');
Assert.ThatBool(
	actual := containsResult,
	message := "Contains must return TRUE for empty substring in non-empty string"
).IsTrue();

containsResult := TOF_Core.Strings.Contains(stringToSearchIn := '', stringToFind := '');
Assert.ThatBool(
	actual := containsResult,
	message := "Contains must return TRUE for empty substring in empty string"
).IsTrue();

containsResult := TOF_Core.Strings.Contains(stringToSearchIn := '', stringToFind := 'a');
Assert.ThatBool(
	actual := containsResult,
	message := "Contains must return FALSE for non-empty substring in empty string"
).IsFalse();

containsResult := TOF_Core.Strings.Contains(stringToSearchIn := 'Hello, world!', stringToFind := 'xyz');
Assert.ThatBool(
	actual := containsResult,
	message := "Contains must return FALSE when substring is absent"
).IsFalse();

containsResult := TOF_Core.Strings.Contains(stringToSearchIn := 'Hello, world!', stringToFind := 'hello');
Assert.ThatBool(
	actual := containsResult,
	message := "Contains must be case-sensitive"
).IsFalse();

containsResult := TOF_Core.Strings.Contains(stringToSearchIn := 'abc', stringToFind := 'abcdef');
Assert.ThatBool(
	actual := containsResult,
	message := "Contains must return FALSE when substring is longer than source"
).IsFalse();

containsResult := TOF_Core.Strings.Contains(stringToSearchIn := 'aaab', stringToFind := 'aab');
Assert.ThatBool(
	actual := containsResult,
	message := "Contains must restart after a partially matching prefix"
).IsTrue();
END_METHOD

//! <summary>Borrows the concrete class name. Callers must not modify it.</summary>
{attribute 'monitoring' := 'call'}
PROPERTY ClassName : REFERENCE TO STRING
GET
ClassName REF= _ClassName;
END_GET
END_PROPERTY

//! <summary>Borrows the compiler-initialized namespace name. Callers must not modify it.</summary>
{attribute 'monitoring' := 'call'}
PROPERTY NamespaceName : REFERENCE TO STRING
GET
NamespaceName REF= CurrentNamespace.Name;
END_GET
END_PROPERTY

//! <summary>Reports the concrete instance size in bytes.</summary>
{attribute 'monitoring' := 'call'}
PROPERTY SelfSize : ULINT
GET
SelfSize := XSIZEOF(THIS^);
END_GET
END_PROPERTY

END_FUNCTION_BLOCK

// ---- Tests/Strings/String/StringJoinTest.TcPOU
(*
SPDX-FileCopyrightText: c 2026 Oleksandr Tiutyk <trofimich@gmail.com>
SPDX-License-Identifier: MIT
License: https://opensource.org/license/mit
*)

(*!
<summary>Checks full and windowed joining and cursor reuse after insufficient capacity.</summary>
<description>
Uses one task and stays at a stable address while assertions are bound to this instance.
</description>
*)

{attribute 'no_assign'}
{attribute 'no_explicit_call' := 'do not call this function block directly'}
FUNCTION_BLOCK StringJoinTest EXTENDS TOF_Testing.SingleCycleTest
VAR_STAT
	{attribute 'hide'}
	_ClassName : STRING := __POUNAME();
END_VAR
VAR
	_Source : STRING := '123 , , 456, 789 ,0';
	_Splitter : TOF_Core.StringSplittingEnumerator;
END_VAR

(*!
<summary>Checks full and windowed joining and cursor reuse after insufficient capacity.</summary>
<description>
Owns a persistent cursor and its borrowed source. Reset releases the current fragment before the result is reported.
</description>
*)
METHOD PROTECTED ExecuteTest
VAR
	separator : STRING := ',';
	joined : STRING := 'old target';
	shortTarget : STRING(2);
	accepted : BOOL;
END_VAR
_Splitter := TOF_Core.Strings.CreateSplitter(sourceString := _Source, separator := separator);
TOF_Core.Strings.Join(targetString := joined, separator := separator, sourceEnumerator := _Splitter);
Assert.ThatBool(
	actual := joined = _Source,
	message := "Unrestricted Join must reconstruct all fragments including their whitespace"
).IsTrue();

_Splitter.Reset();
_Splitter := TOF_Core.Strings.CreateSplitter(
	sourceString := _Source,
	separator := separator,
	maxCount := 3,
	trimEntries := TRUE,
	removeEmptyEntries := TRUE
);
TOF_Core.Strings.Join(
	targetString := joined,
	separator := separator,
	sourceEnumerator := _Splitter,
	startIndex := 1,
	count := 2
);
Assert.ThatBool(
	actual := joined = '456,789',
	message := "The requested window must contain fragments 1 and 2"
).IsTrue();

_Splitter.Reset();
accepted := TOF_Core.Strings.TryJoin(targetString := shortTarget, separator := separator, sourceEnumerator := _Splitter);
Assert.ThatBool(
	actual := accepted,
	message := "TryJoin must reject a target too small for the first fragment"
).IsFalse();

_Splitter.Reset();
accepted := TOF_Core.Strings.TryJoin(
	targetString := joined,
	separator := separator,
	sourceEnumerator := _Splitter,
	count := 1
);
Assert.ThatBool(
	actual := accepted AND_THEN joined = '123',
	message := "After Reset, TryJoin must restart and replace the old target text"
).IsTrue();
END_METHOD

(*!
<summary>Resets the splitter and releases any active fragment before reporting.</summary>
<description>
Safe after partial initialization and after explicit cleanup in the scenario.
</description>
*)
METHOD PROTECTED AfterTest
_Splitter.Reset();
END_METHOD

//! <summary>Borrows the concrete class name. Callers must not modify it.</summary>
{attribute 'monitoring' := 'call'}
PROPERTY ClassName : REFERENCE TO STRING
GET
ClassName REF= _ClassName;
END_GET
END_PROPERTY

//! <summary>Borrows the compiler-initialized namespace name. Callers must not modify it.</summary>
{attribute 'monitoring' := 'call'}
PROPERTY NamespaceName : REFERENCE TO STRING
GET
NamespaceName REF= CurrentNamespace.Name;
END_GET
END_PROPERTY

//! <summary>Reports the concrete instance size in bytes.</summary>
{attribute 'monitoring' := 'call'}
PROPERTY SelfSize : ULINT
GET
SelfSize := XSIZEOF(THIS^);
END_GET
END_PROPERTY

END_FUNCTION_BLOCK

// ---- Tests/Strings/String/StringReplacementTest.TcPOU
(*
SPDX-FileCopyrightText: c 2026 Oleksandr Tiutyk <trofimich@gmail.com>
SPDX-License-Identifier: MIT
License: https://opensource.org/license/mit
*)

(*!
<summary>Checks in-place replacements, counts, limits and partial capacity failure.</summary>
<description>
Uses one task and stays at a stable address while assertions are bound to this instance.
</description>
*)

{attribute 'no_assign'}
{attribute 'no_explicit_call' := 'do not call this function block directly'}
FUNCTION_BLOCK StringReplacementTest EXTENDS TOF_Testing.SingleCycleTest
VAR_STAT
	{attribute 'hide'}
	_ClassName : STRING := __POUNAME();
END_VAR

(*!
<summary>Checks in-place replacements, counts, limits and partial capacity failure.</summary>
<description>
Uses caller-owned buffers with known capacities. A failed next replacement must leave earlier matches applied.
</description>
*)
METHOD PROTECTED ExecuteTest
VAR
	text : STRING(18);
	
	replacementCount : UINT;
	result : BOOL;
END_VAR
text := 'abcd_abcd_abcd';
TOF_Core.Strings.ReplaceInSource(
	sourceString := text,
	oldSubstring := 'bc',
	newSubstring := '0',
	replacementCount => replacementCount
);
Assert.ThatBool(
	actual := text = 'a0d_a0d_a0d',
	message := "Shrink must produce the expected text"
).IsTrue();
Assert.ThatUInt(
	actual := replacementCount,
	message := "Shrink must produce the expected count"
).ToBe(expected := 3);

text := 'abcd_abcd_abcd';
TOF_Core.Strings.ReplaceInSource(
	sourceString := text,
	oldSubstring := 'bc',
	newSubstring := '123',
	replacementCount => replacementCount
);
Assert.ThatBool(
	actual := text = 'a123d_a123d_a123d',
	message := "Grow must produce the expected text"
).IsTrue();
Assert.ThatUInt(
	actual := replacementCount,
	message := "Grow must produce the expected count"
).ToBe(expected := 3);

text := 'abcd_abcd_abcd';
result := TOF_Core.Strings.TryReplaceInSource(
	sourceString := text,
	oldSubstring := 'bc',
	newSubstring := '0',
	replacementCount => replacementCount
);
Assert.ThatBool(
	actual := result,
	message := "Try shrink must produce the expected status"
).IsTrue();
Assert.ThatBool(
	actual := text = 'a0d_a0d_a0d',
	message := "Try shrink must produce the expected text"
).IsTrue();
Assert.ThatUInt(
	actual := replacementCount,
	message := "Try shrink must produce the expected count"
).ToBe(expected := 3);

text := 'abcd_abcd_abcd';
result := TOF_Core.Strings.TryReplaceInSource(
	sourceString := text,
	oldSubstring := 'bc',
	newSubstring := '123',
	maxReplacements := 1,
	skipReplacements := 1,
	replacementCount => replacementCount
);
Assert.ThatBool(
	actual := result,
	message := "Try skip and limit must produce the expected status"
).IsTrue();
Assert.ThatBool(
	actual := text = 'abcd_a123d_abcd',
	message := "Try skip and limit must produce the expected text"
).IsTrue();
Assert.ThatUInt(
	actual := replacementCount,
	message := "Try skip and limit must produce the expected count"
).ToBe(expected := 1);

text := 'abcd_abcd_abcd';
result := TOF_Core.Strings.TryReplaceInSource(
	sourceString := text,
	oldSubstring := 'bc',
	newSubstring := '1234',
	replacementCount => replacementCount
);
Assert.ThatBool(
	actual := result,
	message := "Growth must report failure when the next replacement exceeds capacity"
).IsFalse();
Assert.ThatBool(
	actual := text = 'a1234d_a1234d_abcd',
	message := "Capacity failure must preserve both completed replacements"
).IsTrue();
Assert.ThatUInt(
	actual := replacementCount,
	message := "Capacity failure must report both completed replacements"
).ToBe(expected := UINT#2);

text := 'abcd_abcd';
result := TOF_Core.Strings.TryReplaceInSource(
	sourceString := text,
	oldSubstring := '',
	newSubstring := 'ignore',
	replacementCount => replacementCount
);
Assert.ThatBool(
	actual := result AND_THEN text = 'abcd_abcd' AND_THEN replacementCount = 0,
	message := "An empty search must succeed without modifying text or reporting replacements"
).IsTrue();

result := TOF_Core.Strings.TryReplaceInSource(
	sourceString := text,
	oldSubstring := 'bc',
	newSubstring := '',
	replacementCount => replacementCount
);
Assert.ThatBool(
	actual := result AND_THEN text = 'ad_ad' AND_THEN replacementCount = 2,
	message := "An empty replacement must delete both matching substrings"
).IsTrue();
END_METHOD

//! <summary>Borrows the concrete class name. Callers must not modify it.</summary>
{attribute 'monitoring' := 'call'}
PROPERTY ClassName : REFERENCE TO STRING
GET
ClassName REF= _ClassName;
END_GET
END_PROPERTY

//! <summary>Borrows the compiler-initialized namespace name. Callers must not modify it.</summary>
{attribute 'monitoring' := 'call'}
PROPERTY NamespaceName : REFERENCE TO STRING
GET
NamespaceName REF= CurrentNamespace.Name;
END_GET
END_PROPERTY

//! <summary>Reports the concrete instance size in bytes.</summary>
{attribute 'monitoring' := 'call'}
PROPERTY SelfSize : ULINT
GET
SelfSize := XSIZEOF(THIS^);
END_GET
END_PROPERTY

END_FUNCTION_BLOCK

// ---- Tests/Strings/String/StringSplitTest.TcPOU
(*
SPDX-FileCopyrightText: c 2026 Oleksandr Tiutyk <trofimich@gmail.com>
SPDX-License-Identifier: MIT
License: https://opensource.org/license/mit
*)

(*!
<summary>Checks split fragments, end-of-iteration behavior and cursor restart.</summary>
<description>
Uses one task and stays at a stable address while assertions are bound to this instance.
</description>
*)

{attribute 'no_assign'}
{attribute 'no_explicit_call' := 'do not call this function block directly'}
FUNCTION_BLOCK StringSplitTest EXTENDS TOF_Testing.SingleCycleTest
VAR_STAT
	{attribute 'hide'}
	_ClassName : STRING := __POUNAME();
END_VAR
VAR
	_Source : STRING := '123 , , 456, 789 ,0,';
	_Splitter : TOF_Core.StringSplittingEnumerator;
END_VAR

(*!
<summary>Checks split fragments, end-of-iteration behavior and cursor restart.</summary>
<description>
Owns a persistent cursor and its borrowed source. Reset releases the current fragment before the result is reported.
</description>
*)
METHOD PROTECTED ExecuteTest
VAR
	separator : STRING := ',';
	allFragments : ARRAY [0..5] OF STRING := ['123 ', ' ', ' 456', ' 789 ', '0', ''];
	selectedFragments : ARRAY [0..2] OF STRING := ['123', '456', '789'];
	entry : REFERENCE TO STRING;
	advanced : BOOL;
END_VAR
_Splitter := TOF_Core.Strings.CreateSplitter(sourceString := _Source, separator := separator);
assertFragments(expected := allFragments, scenario := "Unrestricted split");

_Splitter.Reset();
_Splitter := TOF_Core.Strings.CreateSplitter(
	sourceString := _Source,
	separator := separator,
	maxCount := 3,
	trimEntries := TRUE,
	removeEmptyEntries := TRUE
);
assertFragments(expected := selectedFragments, scenario := "Trimmed split limited to three");

_Splitter.Reset();
entry REF= _Splitter.CurrentEntry;
Assert.ThatBool(
	actual := __ISVALIDREF(entry),
	message := "Reset must leave CurrentEntry invalid until the next successful move"
).IsFalse();

advanced := _Splitter.MoveNext();
entry REF= _Splitter.CurrentEntry;
Assert.ThatBool(
	actual := advanced AND_THEN __ISVALIDREF(entry) AND_THEN entry = '123',
	message := "After Reset the first trimmed fragment must be available again"
).IsTrue();
END_METHOD

(*!
<summary>Checks the requested finite sequence and detects trailing fragments or a stale current reference.</summary>
<param name="expected">Expected fragments in order.</param>
<param name="scenario">Cursor configuration included in failure messages.</param>
*)
METHOD PRIVATE assertFragments
VAR_IN_OUT CONSTANT
	expected : ARRAY [*] OF STRING;
END_VAR
VAR_INPUT
	scenario : WSTRING(80);
END_VAR
VAR
	entry : REFERENCE TO STRING;
	i : DINT;
	advanced : BOOL;
	fragmentLabel : WSTRING(255);
END_VAR
FOR i := LOWER_BOUND(expected, 1) TO UPPER_BOUND(expected, 1) DO
	fragmentLabel := Tc2_Utilities.WCONCAT(STR1 := scenario, STR2 := " fragment ");
	fragmentLabel := Tc2_Utilities.WCONCAT(STR1 := fragmentLabel, STR2 := TO_WSTRING(i));
	advanced := _Splitter.MoveNext();
	Assert.ThatBool(actual := advanced, message := fragmentLabel).IsTrue();

	IF NOT advanced THEN
		RETURN;
	END_IF

	entry REF= _Splitter.CurrentEntry;
	Assert.ThatBool(actual := __ISVALIDREF(entry) AND_THEN entry = expected[i], message := fragmentLabel).IsTrue();
END_FOR

advanced := _Splitter.MoveNext();
Assert.ThatBool(
	actual := advanced,
	message := Tc2_Utilities.WCONCAT(STR1 := "Unexpected extra fragment in ", STR2 := scenario)
).IsFalse();

IF advanced THEN
	RETURN;
END_IF

entry REF= _Splitter.CurrentEntry;
Assert.ThatBool(actual := __ISVALIDREF(entry), message := "End of iteration must invalidate CurrentEntry").IsFalse();
advanced := _Splitter.MoveNext();
Assert.ThatBool(actual := advanced, message := "An exhausted splitter must stay exhausted").IsFalse();
END_METHOD

(*!
<summary>Resets the splitter and releases any active fragment before reporting.</summary>
<description>
Safe after partial initialization and after explicit cleanup in the scenario.
</description>
*)
METHOD PROTECTED AfterTest
_Splitter.Reset();
END_METHOD

//! <summary>Borrows the concrete class name. Callers must not modify it.</summary>
{attribute 'monitoring' := 'call'}
PROPERTY ClassName : REFERENCE TO STRING
GET
ClassName REF= _ClassName;
END_GET
END_PROPERTY

//! <summary>Borrows the compiler-initialized namespace name. Callers must not modify it.</summary>
{attribute 'monitoring' := 'call'}
PROPERTY NamespaceName : REFERENCE TO STRING
GET
NamespaceName REF= CurrentNamespace.Name;
END_GET
END_PROPERTY

//! <summary>Reports the concrete instance size in bytes.</summary>
{attribute 'monitoring' := 'call'}
PROPERTY SelfSize : ULINT
GET
SelfSize := XSIZEOF(THIS^);
END_GET
END_PROPERTY

END_FUNCTION_BLOCK

// ---- Tests/Strings/String/StringTrimTest.TcPOU
(*
SPDX-FileCopyrightText: c 2026 Oleksandr Tiutyk <trofimich@gmail.com>
SPDX-License-Identifier: MIT
License: https://opensource.org/license/mit
*)

(*!
<summary>Checks trimming direction, custom characters and complete removal.</summary>
<description>
Uses one task and stays at a stable address while assertions are bound to this instance.
</description>
*)

{attribute 'no_assign'}
{attribute 'no_explicit_call' := 'do not call this function block directly'}
FUNCTION_BLOCK StringTrimTest EXTENDS TOF_Testing.SingleCycleTest
VAR_STAT
	{attribute 'hide'}
	_ClassName : STRING := __POUNAME();
END_VAR

(*!
<summary>Checks trimming direction, custom characters and complete removal.</summary>
*)
METHOD PROTECTED ExecuteTest
VAR
	text : STRING;
END_VAR
text := '  123   ';
TOF_Core.Strings.TrimChar(stringToTrim := text, trimMode := TOF_Core.TRIM_MODE.LEFT_AND_RIGHT);
Assert.ThatBool(
	actual := text = '123',
	message := "TrimChar must apply LEFT_AND_RIGHT exactly"
).IsTrue();

text := '  123   ';
TOF_Core.Strings.TrimChar(stringToTrim := text, trimMode := TOF_Core.TRIM_MODE.LEFT);
Assert.ThatBool(
	actual := text = '123   ',
	message := "TrimChar must apply LEFT exactly"
).IsTrue();

text := '  123   ';
TOF_Core.Strings.TrimChar(stringToTrim := text, trimMode := TOF_Core.TRIM_MODE.RIGHT);
Assert.ThatBool(
	actual := text = '  123',
	message := "TrimChar must apply RIGHT exactly"
).IsTrue();

text := '**a*b**';
TOF_Core.Strings.TrimChar(stringToTrim := text, trimMode := TOF_Core.TRIM_MODE.LEFT_AND_RIGHT, trimChar := '*');
Assert.ThatBool(
	actual := text = 'a*b',
	message := "Trimming a custom character must preserve an internal match"
).IsTrue();

